LIN {X 0,Y 474.559,Z 355.992,A -85,B 0,C 180,E1 -7422.941,E2 -7422.941} C_VEL
LIN {X 0,Y 474.594,Z 355.995,A -85,B 0,C 180,E1 -7425.896,E2 -7425.896} C_VEL
LIN {X 0,Y 474.593,Z 355.988,A -85,B 0,C 180,E1 -7429.046,E2 -7429.046} C_VEL
LIN {X 0,Y 474.585,Z 355.996,A -85,B 0,C 180,E1 -7431.708,E2 -7431.708} C_VEL
LIN {X 0,Y 474.612,Z 355.985,A -85,B 0,C 180,E1 -7434.727,E2 -7434.727} C_VEL
LIN {X 0,Y 474.63,Z 355.992,A -85,B 0,C 180,E1 -7437.789,E2 -7437.789} C_VEL
LIN {X 0,Y 474.593,Z 355.988,A -85,B 0,C 180,E1 -7440.892,E2 -7440.892} C_VEL
LIN {X 0,Y 474.579,Z 355.996,A -85,B 0,C 180,E1 -7443.625,E2 -7443.625} C_VEL
LIN {X 0,Y 474.632,Z 355.983,A -85,B 0,C 180,E1 -7446.644,E2 -7446.644} C_VEL
LIN {X 0,Y 474.65,Z 355.984,A -85,B 0,C 180,E1 -7450.091,E2 -7450.091} C_VEL
LIN {X 0,Y 474.642,Z 355.986,A -85,B 0,C 180,E1 -7451.641,E2 -7451.641} C_VEL
LIN {X 0,Y 473.97,Z 356.072,A -85,B 0,C 180,E1 -7452.35,E2 -7452.35} C_VEL
LIN {X 0,Y 471.124,Z 356.427,A -85,B 0,C 180,E1 -7453.501,E2 -7453.501} C_VEL
LIN {X 0,Y 468.718,Z 356.724,A -85,B 0,C 180,E1 -7454.429,E2 -7454.429} C_VEL
LIN {X 0,Y 467.679,Z 356.851,A -85,B 0,C 180,E1 -7455.147,E2 -7455.147} C_VEL
LIN {X 0,Y 467.592,Z 356.861,A -85,B 0,C 180,E1 -7455.389,E2 -7455.389} C_VEL
LIN {X 0,Y 467.65,Z 356.853,A -85,B 0,C 180,E1 -7458.735,E2 -7458.735} C_VEL
LIN {X 0,Y 467.658,Z 356.855,A -85,B 0,C 180,E1 -7461.358,E2 -7461.358} C_VEL
LIN {X 0,Y 467.705,Z 356.85,A -85,B 0,C 180,E1 -7463.963,E2 -7463.963} C_VEL
LIN {X 0,Y 467.816,Z 356.837,A -85,B 0,C 180,E1 -7467.418,E2 -7467.418} C_VEL
LIN {X 0,Y 467.853,Z 356.831,A -85,B 0,C 180,E1 -7470.001,E2 -7470.001} C_VEL
LIN {X 0,Y 467.818,Z 356.832,A -85,B 0,C 180,E1 -7472.584,E2 -7472.584} C_VEL
LIN {X 0,Y 467.708,Z 356.848,A -85,B 0,C 180,E1 -7476.039,E2 -7476.039} C_VEL
LIN {X 0,Y 467.671,Z 356.85,A -85,B 0,C 180,E1 -7478.644,E2 -7478.644} C_VEL
LIN {X 0,Y 467.662,Z 356.853,A -85,B 0,C 180,E1 -7482.146,E2 -7482.146} C_VEL
LIN {X 0,Y 467.618,Z 356.864,A -85,B 0,C 180,E1 -7485.697,E2 -7485.697} C_VEL
LIN {X 0,Y 467.626,Z 356.86,A -85,B 0,C 180,E1 -7489.309,E2 -7489.309} C_VEL
LIN {X 0,Y 467.54,Z 356.868,A -85,B 0,C 180,E1 -7492.075,E2 -7492.075} C_VEL
LIN {X 0,Y 467.565,Z 356.864,A -85,B 0,C 180,E1 -7494.891,E2 -7494.891} C_VEL
LIN {X 0,Y 467.552,Z 356.87,A -85,B 0,C 180,E1 -7497.774,E2 -7497.774} C_VEL
LIN {X 0,Y 467.572,Z 356.865,A -85,B 0,C 180,E1 -7501.045,E2 -7501.045} C_VEL
LIN {X 0,Y 467.593,Z 356.86,A -85,B 0,C 180,E1 -7504.242,E2 -7504.242} C_VEL
LIN {X 0,Y 467.549,Z 356.873,A -85,B 0,C 180,E1 -7507.186,E2 -7507.186} C_VEL
LIN {X 0,Y 467.576,Z 356.867,A -85,B 0,C 180,E1 -7510.266,E2 -7510.266} C_VEL
LIN {X 0,Y 467.567,Z 356.868,A -85,B 0,C 180,E1 -7512.564,E2 -7512.564} C_VEL
LIN {X 0,Y 467.561,Z 356.872,A -85,B 0,C 180,E1 -7514.121,E2 -7514.121} C_VEL
LIN {X 0,Y 470.952,Z 371.96,A -85,B 0,C 180,E1 -7516.951,E2 -7516.951} C_VEL
LIN {X 0,Y 474.676,Z 387.334,A -85,B 0,C 180,E1 -7517.428,E2 -7517.428} C_VEL
LIN {X 0,Y 475.85,Z 392.656,A -85,B 0,C 180,E1 -7517.582,E2 -7517.582} C_VEL
LIN {X 0,Y 473.727,Z 537.942,A -85,B 0,C 180,E1 -7519.999,E2 -7519.999} C_VEL
LIN {X 0,Y 473.257,Z 553.297,A -85,B 0,C 180,E1 -7520.424,E2 -7520.424} C_VEL
LIN {X 0,Y 472.684,Z 567.565,A -85,B 0,C 180,E1 -7520.982,E2 -7520.982} C_VEL
LIN {X 0,Y 471.947,Z 582.804,A -85,B 0,C 180,E1 -7521.773,E2 -7521.773} C_VEL
LIN {X 0,Y 471.223,Z 596.937,A -85,B 0,C 180,E1 -7522.706,E2 -7522.706} C_VEL
LIN {X 0,Y 470.38,Z 610.271,A -85,B 0,C 180,E1 -7523.788,E2 -7523.788} C_VEL
LIN {X 0,Y 469.675,Z 622.164,A -85,B 0,C 180,E1 -7524.954,E2 -7524.954} C_VEL
LIN {X 0,Y 468.906,Z 633.77,A -85,B 0,C 180,E1 -7526.319,E2 -7526.319} C_VEL
LIN {X 0,Y 468.273,Z 644.266,A -85,B 0,C 180,E1 -7527.805,E2 -7527.805} C_VEL
LIN {X 0,Y 467.78,Z 652.986,A -85,B 0,C 180,E1 -7529.281,E2 -7529.281} C_VEL
LIN {X 0,Y 467.331,Z 661.21,A -85,B 0,C 180,E1 -7530.971,E2 -7530.971} C_VEL
LIN {X 0,Y 467.022,Z 667.684,A -85,B 0,C 180,E1 -7532.607,E2 -7532.607} C_VEL
LIN {X 0,Y 466.836,Z 672.428,A -85,B 0,C 180,E1 -7534.114,E2 -7534.114} C_VEL
LIN {X 0,Y 466.715,Z 676.016,A -85,B 0,C 180,E1 -7535.537,E2 -7535.537} C_VEL
LIN {X 0,Y 466.612,Z 678.697,A -85,B 0,C 180,E1 -7536.945,E2 -7536.945} C_VEL
LIN {X 0,Y 466.538,Z 681.023,A -85,B 0,C 180,E1 -7538.805,E2 -7538.805} C_VEL
LIN {X 0,Y 466.523,Z 681.987,A -85,B 0,C 180,E1 -7540.645,E2 -7540.645} C_VEL
LIN {X 0,Y 466.534,Z 681.648,A -85,B 0,C 180,E1 -7542.465,E2 -7542.465} C_VEL
LIN {X 0,Y 466.539,Z 680.045,A -85,B 0,C 180,E1 -7544.267,E2 -7544.267} C_VEL
LIN {X 0,Y 466.613,Z 677.173,A -85,B 0,C 180,E1 -7546.055,E2 -7546.055} C_VEL
LIN {X 0,Y 466.856,Z 672.982,A -85,B 0,C 180,E1 -7547.833,E2 -7547.833} C_VEL
LIN {X 0,Y 467.035,Z 667.435,A -85,B 0,C 180,E1 -7549.596,E2 -7549.596} C_VEL
LIN {X 0,Y 467.402,Z 660.369,A -85,B 0,C 180,E1 -7551.352,E2 -7551.352} C_VEL
LIN {X 0,Y 467.801,Z 653.127,A -85,B 0,C 180,E1 -7552.824,E2 -7552.824} C_VEL
LIN {X 0,Y 468.295,Z 643.765,A -85,B 0,C 180,E1 -7554.402,E2 -7554.402} C_VEL
LIN {X 0,Y 468.97,Z 632.863,A -85,B 0,C 180,E1 -7555.918,E2 -7555.918} C_VEL
LIN {X 0,Y 469.723,Z 621.677,A -85,B 0,C 180,E1 -7557.213,E2 -7557.213} C_VEL
LIN {X 0,Y 470.482,Z 609.45,A -85,B 0,C 180,E1 -7558.395,E2 -7558.395} C_VEL
LIN {X 0,Y 471.319,Z 596.43,A -85,B 0,C 180,E1 -7559.435,E2 -7559.435} C_VEL
LIN {X 0,Y 472.012,Z 582.911,A -85,B 0,C 180,E1 -7560.32,E2 -7560.32} C_VEL
LIN {X 0,Y 472.671,Z 568.576,A -85,B 0,C 180,E1 -7561.065,E2 -7561.065} C_VEL
LIN {X 0,Y 473.286,Z 552.999,A -85,B 0,C 180,E1 -7561.675,E2 -7561.675} C_VEL
LIN {X 0,Y 473.757,Z 537.298,A -85,B 0,C 180,E1 -7562.099,E2 -7562.099} C_VEL
LIN {X 0,Y 476.168,Z 392.734,A -85,B 0,C 180,E1 -7564.596,E2 -7564.596} C_VEL
LIN {X 0,Y 472.006,Z 375.11,A -85,B 0,C 180,E1 -7565.179,E2 -7565.179} C_VEL
LIN {X 0,Y 471.448,Z 373.4,A -85,B 0,C 180,E1 -7565.265,E2 -7565.265} C_VEL
LIN {X 0,Y 469.366,Z 363.6,A -85,B 0,C 180,E1 -7567.194,E2 -7567.194} C_VEL
LIN {X 0,Y 467.682,Z 356.858,A -85,B 0,C 180,E1 -7568.613,E2 -7568.613} C_VEL
LIN {X 0,Y 467.661,Z 356.858,A -85,B 0,C 180,E1 -7572.145,E2 -7572.145} C_VEL
LIN {X 0,Y 467.643,Z 356.859,A -85,B 0,C 180,E1 -7575.695,E2 -7575.695} C_VEL
LIN {X 0,Y 467.626,Z 356.86,A -85,B 0,C 180,E1 -7579.307,E2 -7579.307} C_VEL
LIN {X 0,Y 467.539,Z 356.873,A -85,B 0,C 180,E1 -7582.073,E2 -7582.073} C_VEL
LIN {X 0,Y 467.559,Z 356.867,A -85,B 0,C 180,E1 -7584.89,E2 -7584.89} C_VEL
LIN {X 0,Y 467.548,Z 356.871,A -85,B 0,C 180,E1 -7587.773,E2 -7587.773} C_VEL
LIN {X 0,Y 467.55,Z 356.867,A -85,B 0,C 180,E1 -7591.04,E2 -7591.04} C_VEL
LIN {X 0,Y 467.578,Z 356.868,A -85,B 0,C 180,E1 -7594.239,E2 -7594.239} C_VEL
LIN {X 0,Y 467.517,Z 356.872,A -85,B 0,C 180,E1 -7597.18,E2 -7597.18} C_VEL
LIN {X 0,Y 467.541,Z 356.872,A -85,B 0,C 180,E1 -7600.268,E2 -7600.268} C_VEL
LIN {X 0,Y 467.519,Z 356.873,A -85,B 0,C 180,E1 -7602.568,E2 -7602.568} C_VEL
LIN {X 0,Y 467.564,Z 356.864,A -85,B 0,C 180,E1 -7605.051,E2 -7605.051} C_VEL
LIN {X 0,Y 467.552,Z 356.867,A -85,B 0,C 180,E1 -7608.727,E2 -7608.727} C_VEL
LIN {X 0,Y 467.539,Z 356.875,A -85,B 0,C 180,E1 -7611.952,E2 -7611.952} C_VEL
LIN {X 0,Y 467.541,Z 356.873,A -85,B 0,C 180,E1 -7615.164,E2 -7615.164} C_VEL
LIN {X 0,Y 467.551,Z 356.877,A -85,B 0,C 180,E1 -7618.256,E2 -7618.256} C_VEL
LIN {X 0,Y 467.609,Z 356.988,A -85,B 0,C 180,E1 -7619.362,E2 -7619.362} C_VEL
LIN {X 0,Y 470.846,Z 369.937,A -85,B 0,C 180,E1 -7621.721,E2 -7621.721} C_VEL
LIN {X 0,Y 472.31,Z 377.176,A -85,B 0,C 180,E1 -7622.965,E2 -7622.965} C_VEL
LIN {X 0,Y 471.285,Z 396.039,A -85,B 0,C 180,E1 -7625.777,E2 -7625.777} C_VEL
LIN {X 0,Y 475.861,Z 420.157,A -85,B 0,C 180,E1 -7626.498,E2 -7626.498} C_VEL
LIN {X 0,Y 474.004,Z 533.469,A -85,B 0,C 180,E1 -7628.442,E2 -7628.442} C_VEL
LIN {X 0,Y 473.478,Z 564.563,A -85,B 0,C 180,E1 -7628.987,E2 -7628.987} C_VEL
LIN {X 0,Y 472.916,Z 580.082,A -85,B 0,C 180,E1 -7629.429,E2 -7629.429} C_VEL
LIN {X 0,Y 472.302,Z 595.204,A -85,B 0,C 180,E1 -7630.042,E2 -7630.042} C_VEL
LIN {X 0,Y 471.659,Z 608.713,A -85,B 0,C 180,E1 -7630.75,E2 -7630.75} C_VEL
LIN {X 0,Y 470.924,Z 622.125,A -85,B 0,C 180,E1 -7631.622,E2 -7631.622} C_VEL
LIN {X 0,Y 470.114,Z 634.534,A -85,B 0,C 180,E1 -7632.602,E2 -7632.602} C_VEL
LIN {X 0,Y 469.374,Z 647.182,A -85,B 0,C 180,E1 -7633.806,E2 -7633.806} C_VEL
LIN {X 0,Y 468.596,Z 659.56,A -85,B 0,C 180,E1 -7635.227,E2 -7635.227} C_VEL
LIN {X 0,Y 468.049,Z 669.126,A -85,B 0,C 180,E1 -7636.54,E2 -7636.54} C_VEL
LIN {X 0,Y 467.526,Z 678.506,A -85,B 0,C 180,E1 -7638.07,E2 -7638.07} C_VEL
LIN {X 0,Y 467.224,Z 686.288,A -85,B 0,C 180,E1 -7639.6,E2 -7639.6} C_VEL
LIN {X 0,Y 466.907,Z 693.544,A -85,B 0,C 180,E1 -7641.342,E2 -7641.342} C_VEL
LIN {X 0,Y 466.745,Z 699.247,A -85,B 0,C 180,E1 -7643.08,E2 -7643.08} C_VEL
LIN {X 0,Y 466.686,Z 703.56,A -85,B 0,C 180,E1 -7644.815,E2 -7644.815} C_VEL
LIN {X 0,Y 466.639,Z 706.587,A -85,B 0,C 180,E1 -7646.545,E2 -7646.545} C_VEL
LIN {X 0,Y 466.628,Z 708.398,A -85,B 0,C 180,E1 -7648.273,E2 -7648.273} C_VEL
LIN {X 0,Y 466.595,Z 709.029,A -85,B 0,C 180,E1 -7649.999,E2 -7649.999} C_VEL
LIN {X 0,Y 466.628,Z 708.435,A -85,B 0,C 180,E1 -7651.725,E2 -7651.725} C_VEL
LIN {X 0,Y 466.67,Z 706.662,A -85,B 0,C 180,E1 -7653.452,E2 -7653.452} C_VEL
LIN {X 0,Y 466.69,Z 703.683,A -85,B 0,C 180,E1 -7655.183,E2 -7655.183} C_VEL
LIN {X 0,Y 466.82,Z 699.43,A -85,B 0,C 180,E1 -7656.916,E2 -7656.916} C_VEL
LIN {X 0,Y 466.933,Z 693.785,A -85,B 0,C 180,E1 -7658.655,E2 -7658.655} C_VEL
LIN {X 0,Y 467.222,Z 686.598,A -85,B 0,C 180,E1 -7660.398,E2 -7660.398} C_VEL
LIN {X 0,Y 467.601,Z 678.901,A -85,B 0,C 180,E1 -7661.925,E2 -7661.925} C_VEL
LIN {X 0,Y 468.081,Z 669.621,A -85,B 0,C 180,E1 -7663.456,E2 -7663.456} C_VEL
LIN {X 0,Y 468.648,Z 660.149,A -85,B 0,C 180,E1 -7664.768,E2 -7664.768} C_VEL
LIN {X 0,Y 469.455,Z 647.921,A -85,B 0,C 180,E1 -7666.189,E2 -7666.189} C_VEL
LIN {X 0,Y 470.178,Z 635.42,A -85,B 0,C 180,E1 -7667.393,E2 -7667.393} C_VEL
LIN {X 0,Y 470.931,Z 623.112,A -85,B 0,C 180,E1 -7668.375,E2 -7668.375} C_VEL
LIN {X 0,Y 471.738,Z 609.861,A -85,B 0,C 180,E1 -7669.244,E2 -7669.244} C_VEL
LIN {X 0,Y 472.39,Z 596.536,A -85,B 0,C 180,E1 -7669.952,E2 -7669.952} C_VEL
LIN {X 0,Y 473.025,Z 581.741,A -85,B 0,C 180,E1 -7670.56,E2 -7670.56} C_VEL
LIN {X 0,Y 473.553,Z 566.453,A -85,B 0,C 180,E1 -7671.007,E2 -7671.007} C_VEL
LIN {X 0,Y 473.94,Z 543.805,A -85,B 0,C 180,E1 -7671.416,E2 -7671.416} C_VEL
LIN {X 0,Y 475.645,Z 419.81,A -85,B 0,C 180,E1 -7673.463,E2 -7673.463} C_VEL
LIN {X 0,Y 471.258,Z 396.949,A -85,B 0,C 180,E1 -7674.105,E2 -7674.105} C_VEL
LIN {X 0,Y 472.297,Z 378.855,A -85,B 0,C 180,E1 -7676.77,E2 -7676.77} C_VEL
LIN {X 0,Y 472.051,Z 375.647,A -85,B 0,C 180,E1 -7677.27,E2 -7677.27} C_VEL
LIN {X 0,Y 468.726,Z 361.5,A -85,B 0,C 180,E1 -7679.654,E2 -7679.654} C_VEL
LIN {X 0,Y 467.582,Z 356.868,A -85,B 0,C 180,E1 -7680.481,E2 -7680.481} C_VEL
LIN {X 0,Y 467.561,Z 356.869,A -85,B 0,C 180,E1 -7683.788,E2 -7683.788} C_VEL
LIN {X 0,Y 467.503,Z 356.874,A -85,B 0,C 180,E1 -7686.963,E2 -7686.963} C_VEL
LIN {X 0,Y 467.551,Z 356.871,A -85,B 0,C 180,E1 -7689.95,E2 -7689.95} C_VEL
LIN {X 0,Y 467.532,Z 356.871,A -85,B 0,C 180,E1 -7692.564,E2 -7692.564} C_VEL
LIN {X 0,Y 467.553,Z 356.865,A -85,B 0,C 180,E1 -7695.051,E2 -7695.051} C_VEL
LIN {X 0,Y 467.548,Z 356.867,A -85,B 0,C 180,E1 -7698.725,E2 -7698.725} C_VEL
LIN {X 0,Y 467.528,Z 356.873,A -85,B 0,C 180,E1 -7701.952,E2 -7701.952} C_VEL
LIN {X 0,Y 467.544,Z 356.866,A -85,B 0,C 180,E1 -7705.166,E2 -7705.166} C_VEL
LIN {X 0,Y 467.568,Z 356.87,A -85,B 0,C 180,E1 -7708.259,E2 -7708.259} C_VEL
LIN {X 0,Y 467.529,Z 356.868,A -85,B 0,C 180,E1 -7711.247,E2 -7711.247} C_VEL
LIN {X 0,Y 467.563,Z 356.868,A -85,B 0,C 180,E1 -7714.4,E2 -7714.4} C_VEL
LIN {X 0,Y 467.556,Z 356.864,A -85,B 0,C 180,E1 -7716.995,E2 -7716.995} C_VEL
LIN {X 0,Y 467.604,Z 356.863,A -85,B 0,C 180,E1 -7719.777,E2 -7719.777} C_VEL
LIN {X 0,Y 467.55,Z 356.868,A -85,B 0,C 180,E1 -7722.505,E2 -7722.505} C_VEL
LIN {X 0,Y 467.577,Z 356.862,A -85,B 0,C 180,E1 -7725.196,E2 -7725.196} C_VEL
LIN {X 0,Y 467.64,Z 356.859,A -85,B 0,C 180,E1 -7727.854,E2 -7727.854} C_VEL
LIN {X 0,Y 467.641,Z 356.855,A -85,B 0,C 180,E1 -7731.357,E2 -7731.357} C_VEL
LIN {X 0,Y 467.69,Z 356.855,A -85,B 0,C 180,E1 -7733.962,E2 -7733.962} C_VEL
LIN {X 0,Y 467.796,Z 356.836,A -85,B 0,C 180,E1 -7737.417,E2 -7737.417} C_VEL
LIN {X 0,Y 467.833,Z 356.838,A -85,B 0,C 180,E1 -7740,E2 -7740} C_VEL
LIN {X 0,Y 467.796,Z 356.836,A -85,B 0,C 180,E1 -7742.583,E2 -7742.583} C_VEL
LIN {X 0,Y 467.686,Z 356.856,A -85,B 0,C 180,E1 -7746.038,E2 -7746.038} C_VEL
LIN {X 0,Y 467.639,Z 356.855,A -85,B 0,C 180,E1 -7748.644,E2 -7748.644} C_VEL
LIN {X 0,Y 467.633,Z 356.858,A -85,B 0,C 180,E1 -7752.354,E2 -7752.354} C_VEL
LIN {X 0,Y 467.585,Z 356.868,A -85,B 0,C 180,E1 -7755.864,E2 -7755.864} C_VEL
LIN {X 0,Y 467.604,Z 356.86,A -85,B 0,C 180,E1 -7759.309,E2 -7759.309} C_VEL
LIN {X 0,Y 467.516,Z 356.876,A -85,B 0,C 180,E1 -7762.075,E2 -7762.075} C_VEL
LIN {X 0,Y 467.545,Z 356.866,A -85,B 0,C 180,E1 -7764.891,E2 -7764.891} C_VEL
LIN {X 0,Y 467.531,Z 356.874,A -85,B 0,C 180,E1 -7767.775,E2 -7767.775} C_VEL
LIN {X 0,Y 467.553,Z 356.865,A -85,B 0,C 180,E1 -7771.045,E2 -7771.045} C_VEL
LIN {X 0,Y 467.565,Z 356.867,A -85,B 0,C 180,E1 -7774.241,E2 -7774.241} C_VEL
LIN {X 0,Y 467.506,Z 356.871,A -85,B 0,C 180,E1 -7777.183,E2 -7777.183} C_VEL
LIN {X 0,Y 467.546,Z 356.868,A -85,B 0,C 180,E1 -7780.268,E2 -7780.268} C_VEL
LIN {X 0,Y 467.535,Z 356.874,A -85,B 0,C 180,E1 -7783.747,E2 -7783.747} C_VEL
LIN {X 0,Y 467.538,Z 356.869,A -85,B 0,C 180,E1 -7786.256,E2 -7786.256} C_VEL
LIN {X 0,Y 467.549,Z 356.873,A -85,B 0,C 180,E1 -7789.735,E2 -7789.735} C_VEL
LIN {X 0,Y 467.516,Z 356.869,A -85,B 0,C 180,E1 -7792.82,E2 -7792.82} C_VEL
LIN {X 0,Y 467.571,Z 356.871,A -85,B 0,C 180,E1 -7795.762,E2 -7795.762} C_VEL
LIN {X 0,Y 467.561,Z 356.864,A -85,B 0,C 180,E1 -7798.957,E2 -7798.957} C_VEL
LIN {X 0,Y 467.54,Z 356.869,A -85,B 0,C 180,E1 -7802.228,E2 -7802.228} C_VEL
LIN {X 0,Y 467.553,Z 356.866,A -85,B 0,C 180,E1 -7805.112,E2 -7805.112} C_VEL
LIN {X 0,Y 467.533,Z 356.873,A -85,B 0,C 180,E1 -7807.928,E2 -7807.928} C_VEL
LIN {X 0,Y 467.619,Z 356.856,A -85,B 0,C 180,E1 -7810.694,E2 -7810.694} C_VEL
LIN {X 0,Y 467.638,Z 356.856,A -85,B 0,C 180,E1 -7814.306,E2 -7814.306} C_VEL
LIN {X 0,Y 467.592,Z 356.861,A -85,B 0,C 180,E1 -7815.389,E2 -7815.389} C_VEL
LIN {X 0,Y 466.92,Z 356.947,A -85,B 0,C 180,E1 -7816.109,E2 -7816.109} C_VEL
LIN {X 0,Y 464.081,Z 357.3,A -85,B 0,C 180,E1 -7817.277,E2 -7817.277} C_VEL
LIN {X 0,Y 461.684,Z 357.598,A -85,B 0,C 180,E1 -7818.22,E2 -7818.22} C_VEL
LIN {X 0,Y 460.656,Z 357.725,A -85,B 0,C 180,E1 -7818.947,E2 -7818.947} C_VEL
LIN {X 0,Y 460.572,Z 357.736,A -85,B 0,C 180,E1 -7819.194,E2 -7819.194} C_VEL
LIN {X 0,Y 460.665,Z 357.723,A -85,B 0,C 180,E1 -7822.595,E2 -7822.595} C_VEL
LIN {X 0,Y 460.677,Z 357.721,A -85,B 0,C 180,E1 -7824.749,E2 -7824.749} C_VEL
LIN {X 0,Y 460.76,Z 357.715,A -85,B 0,C 180,E1 -7827.379,E2 -7827.379} C_VEL
LIN {X 0,Y 460.822,Z 357.707,A -85,B 0,C 180,E1 -7830.001,E2 -7830.001} C_VEL
LIN {X 0,Y 460.762,Z 357.711,A -85,B 0,C 180,E1 -7832.624,E2 -7832.624} C_VEL
LIN {X 0,Y 460.674,Z 357.724,A -85,B 0,C 180,E1 -7836.132,E2 -7836.132} C_VEL
LIN {X 0,Y 460.622,Z 357.728,A -85,B 0,C 180,E1 -7838.777,E2 -7838.777} C_VEL
LIN {X 0,Y 460.602,Z 357.731,A -85,B 0,C 180,E1 -7842.436,E2 -7842.436} C_VEL
LIN {X 0,Y 460.562,Z 357.739,A -85,B 0,C 180,E1 -7845.979,E2 -7845.979} C_VEL
LIN {X 0,Y 460.572,Z 357.742,A -85,B 0,C 180,E1 -7849.616,E2 -7849.616} C_VEL
LIN {X 0,Y 460.516,Z 357.741,A -85,B 0,C 180,E1 -7852.43,E2 -7852.43} C_VEL
LIN {X 0,Y 460.541,Z 357.743,A -85,B 0,C 180,E1 -7855.794,E2 -7855.794} C_VEL
LIN {X 0,Y 460.526,Z 357.744,A -85,B 0,C 180,E1 -7859.233,E2 -7859.233} C_VEL
LIN {X 0,Y 460.537,Z 357.739,A -85,B 0,C 180,E1 -7862.285,E2 -7862.285} C_VEL
LIN {X 0,Y 460.514,Z 357.749,A -85,B 0,C 180,E1 -7865.446,E2 -7865.446} C_VEL
LIN {X 0,Y 460.511,Z 357.747,A -85,B 0,C 180,E1 -7868.892,E2 -7868.892} C_VEL
LIN {X 0,Y 460.524,Z 357.748,A -85,B 0,C 180,E1 -7871.601,E2 -7871.601} C_VEL
LIN {X 0,Y 460.523,Z 357.748,A -85,B 0,C 180,E1 -7873.827,E2 -7873.827} C_VEL
LIN {X 0,Y 463.793,Z 372.282,A -85,B 0,C 180,E1 -7876.587,E2 -7876.587} C_VEL
LIN {X 0,Y 465.856,Z 378.515,A -85,B 0,C 180,E1 -7876.813,E2 -7876.813} C_VEL
LIN {X 0,Y 469.226,Z 393.41,A -85,B 0,C 180,E1 -7877.256,E2 -7877.256} C_VEL
LIN {X 0,Y 467.185,Z 529.999,A -85,B 0,C 180,E1 -7879.553,E2 -7879.553} C_VEL
LIN {X 0,Y 466.793,Z 546.261,A -85,B 0,C 180,E1 -7879.92,E2 -7879.92} C_VEL
LIN {X 0,Y 466.209,Z 561.626,A -85,B 0,C 180,E1 -7880.448,E2 -7880.448} C_VEL
LIN {X 0,Y 465.578,Z 576.36,A -85,B 0,C 180,E1 -7881.141,E2 -7881.141} C_VEL
LIN {X 0,Y 464.891,Z 589.468,A -85,B 0,C 180,E1 -7881.921,E2 -7881.921} C_VEL
LIN {X 0,Y 463.999,Z 603.248,A -85,B 0,C 180,E1 -7882.933,E2 -7882.933} C_VEL
LIN {X 0,Y 463.243,Z 615.11,A -85,B 0,C 180,E1 -7883.992,E2 -7883.992} C_VEL
LIN {X 0,Y 462.492,Z 625.965,A -85,B 0,C 180,E1 -7885.144,E2 -7885.144} C_VEL
LIN {X 0,Y 461.744,Z 636.861,A -85,B 0,C 180,E1 -7886.513,E2 -7886.513} C_VEL
LIN {X 0,Y 461.153,Z 646.802,A -85,B 0,C 180,E1 -7888.008,E2 -7888.008} C_VEL
LIN {X 0,Y 460.63,Z 655.174,A -85,B 0,C 180,E1 -7889.515,E2 -7889.515} C_VEL
LIN {X 0,Y 460.228,Z 663.103,A -85,B 0,C 180,E1 -7891.247,E2 -7891.247} C_VEL
LIN {X 0,Y 459.941,Z 668.61,A -85,B 0,C 180,E1 -7892.715,E2 -7892.715} C_VEL
LIN {X 0,Y 459.74,Z 673.716,A -85,B 0,C 180,E1 -7894.414,E2 -7894.414} C_VEL
LIN {X 0,Y 459.625,Z 676.526,A -85,B 0,C 180,E1 -7895.616,E2 -7895.616} C_VEL
LIN {X 0,Y 459.453,Z 679.82,A -85,B 0,C 180,E1 -7897.517,E2 -7897.517} C_VEL
LIN {X 0,Y 459.448,Z 681.698,A -85,B 0,C 180,E1 -7899.401,E2 -7899.401} C_VEL
LIN {X 0,Y 459.444,Z 682.236,A -85,B 0,C 180,E1 -7901.262,E2 -7901.262} C_VEL
LIN {X 0,Y 459.428,Z 681.484,A -85,B 0,C 180,E1 -7903.103,E2 -7903.103} C_VEL
LIN {X 0,Y 459.505,Z 679.461,A -85,B 0,C 180,E1 -7904.929,E2 -7904.929} C_VEL
LIN {X 0,Y 459.624,Z 676.139,A -85,B 0,C 180,E1 -7906.74,E2 -7906.74} C_VEL
LIN {X 0,Y 459.823,Z 671.486,A -85,B 0,C 180,E1 -7908.539,E2 -7908.539} C_VEL
LIN {X 0,Y 460.074,Z 665.437,A -85,B 0,C 180,E1 -7910.326,E2 -7910.326} C_VEL
LIN {X 0,Y 460.531,Z 657.824,A -85,B 0,C 180,E1 -7912.105,E2 -7912.105} C_VEL
LIN {X 0,Y 461.003,Z 649.687,A -85,B 0,C 180,E1 -7913.654,E2 -7913.654} C_VEL
LIN {X 0,Y 461.624,Z 639.949,A -85,B 0,C 180,E1 -7915.196,E2 -7915.196} C_VEL
LIN {X 0,Y 462.315,Z 630.001,A -85,B 0,C 180,E1 -7916.514,E2 -7916.514} C_VEL
LIN {X 0,Y 463.062,Z 618.257,A -85,B 0,C 180,E1 -7917.825,E2 -7917.825} C_VEL
LIN {X 0,Y 463.929,Z 605.963,A -85,B 0,C 180,E1 -7918.964,E2 -7918.964} C_VEL
LIN {X 0,Y 464.735,Z 592.437,A -85,B 0,C 180,E1 -7920,E2 -7920} C_VEL
LIN {X 0,Y 465.533,Z 578.411,A -85,B 0,C 180,E1 -7920.865,E2 -7920.865} C_VEL
LIN {X 0,Y 466.188,Z 563.974,A -85,B 0,C 180,E1 -7921.566,E2 -7921.566} C_VEL
LIN {X 0,Y 466.749,Z 549.143,A -85,B 0,C 180,E1 -7922.103,E2 -7922.103} C_VEL
LIN {X 0,Y 467.168,Z 533.927,A -85,B 0,C 180,E1 -7922.479,E2 -7922.479} C_VEL
LIN {X 0,Y 469.596,Z 402.99,A -85,B 0,C 180,E1 -7924.781,E2 -7924.781} C_VEL
LIN {X 0,Y 469.695,Z 393.427,A -85,B 0,C 180,E1 -7924.963,E2 -7924.963} C_VEL
LIN {X 0,Y 465.864,Z 377.43,A -85,B 0,C 180,E1 -7925.518,E2 -7925.518} C_VEL
LIN {X 0,Y 464.428,Z 373.801,A -85,B 0,C 180,E1 -7925.684,E2 -7925.684} C_VEL
LIN {X 0,Y 462.015,Z 363.103,A -85,B 0,C 180,E1 -7927.869,E2 -7927.869} C_VEL
LIN {X 0,Y 460.636,Z 357.734,A -85,B 0,C 180,E1 -7929.052,E2 -7929.052} C_VEL
LIN {X 0,Y 460.602,Z 357.737,A -85,B 0,C 180,E1 -7932.435,E2 -7932.435} C_VEL
LIN {X 0,Y 460.606,Z 357.738,A -85,B 0,C 180,E1 -7935.997,E2 -7935.997} C_VEL
LIN {X 0,Y 460.572,Z 357.739,A -85,B 0,C 180,E1 -7939.615,E2 -7939.615} C_VEL
LIN {X 0,Y 460.515,Z 357.749,A -85,B 0,C 180,E1 -7942.428,E2 -7942.428} C_VEL
LIN {X 0,Y 460.536,Z 357.743,A -85,B 0,C 180,E1 -7945.792,E2 -7945.792} C_VEL
LIN {X 0,Y 460.522,Z 357.744,A -85,B 0,C 180,E1 -7949.232,E2 -7949.232} C_VEL
LIN {X 0,Y 460.521,Z 357.748,A -85,B 0,C 180,E1 -7952.285,E2 -7952.285} C_VEL
LIN {X 0,Y 460.502,Z 357.747,A -85,B 0,C 180,E1 -7955.446,E2 -7955.446} C_VEL
LIN {X 0,Y 460.486,Z 357.747,A -85,B 0,C 180,E1 -7958.887,E2 -7958.887} C_VEL
LIN {X 0,Y 460.497,Z 357.748,A -85,B 0,C 180,E1 -7961.596,E2 -7961.596} C_VEL
LIN {X 0,Y 460.508,Z 357.744,A -85,B 0,C 180,E1 -7964.589,E2 -7964.589} C_VEL
LIN {X 0,Y 460.473,Z 357.752,A -85,B 0,C 180,E1 -7967.812,E2 -7967.812} C_VEL
LIN {X 0,Y 460.477,Z 357.752,A -85,B 0,C 180,E1 -7970.131,E2 -7970.131} C_VEL
LIN {X 0,Y 460.458,Z 357.756,A -85,B 0,C 180,E1 -7973.468,E2 -7973.468} C_VEL
LIN {X 0,Y 460.503,Z 357.753,A -85,B 0,C 180,E1 -7976.672,E2 -7976.672} C_VEL
LIN {X 0,Y 460.519,Z 357.849,A -85,B 0,C 180,E1 -7978.934,E2 -7978.934} C_VEL
LIN {X 0,Y 463.633,Z 369.945,A -85,B 0,C 180,E1 -7981.216,E2 -7981.216} C_VEL
LIN {X 0,Y 465.571,Z 379.235,A -85,B 0,C 180,E1 -7982.853,E2 -7982.853} C_VEL
LIN {X 0,Y 464.544,Z 395.515,A -85,B 0,C 180,E1 -7985.349,E2 -7985.349} C_VEL
LIN {X 0,Y 469.424,Z 421.293,A -85,B 0,C 180,E1 -7986.156,E2 -7986.156} C_VEL
LIN {X 0,Y 467.381,Z 534.879,A -85,B 0,C 180,E1 -7988.15,E2 -7988.15} C_VEL
LIN {X 0,Y 466.861,Z 564.068,A -85,B 0,C 180,E1 -7988.675,E2 -7988.675} C_VEL
LIN {X 0,Y 466.286,Z 579.38,A -85,B 0,C 180,E1 -7989.115,E2 -7989.115} C_VEL
LIN {X 0,Y 465.594,Z 594.743,A -85,B 0,C 180,E1 -7989.742,E2 -7989.742} C_VEL
LIN {X 0,Y 464.896,Z 608.292,A -85,B 0,C 180,E1 -7990.458,E2 -7990.458} C_VEL
LIN {X 0,Y 464.115,Z 621.72,A -85,B 0,C 180,E1 -7991.343,E2 -7991.343} C_VEL
LIN {X 0,Y 463.177,Z 635.394,A -85,B 0,C 180,E1 -7992.447,E2 -7992.447} C_VEL
LIN {X 0,Y 462.399,Z 647.848,A -85,B 0,C 180,E1 -7993.668,E2 -7993.668} C_VEL
LIN {X 0,Y 461.619,Z 659.226,A -85,B 0,C 180,E1 -7994.999,E2 -7994.999} C_VEL
LIN {X 0,Y 461.061,Z 668.805,A -85,B 0,C 180,E1 -7996.332,E2 -7996.332} C_VEL
LIN {X 0,Y 460.504,Z 678.203,A -85,B 0,C 180,E1 -7997.885,E2 -7997.885} C_VEL
LIN {X 0,Y 460.202,Z 686.012,A -85,B 0,C 180,E1 -7999.439,E2 -7999.439} C_VEL
LIN {X 0,Y 459.851,Z 693.286,A -85,B 0,C 180,E1 -8001.208,E2 -8001.208} C_VEL
LIN {X 0,Y 459.665,Z 699.005,A -85,B 0,C 180,E1 -8002.973,E2 -8002.973} C_VEL
LIN {X 0,Y 459.597,Z 703.333,A -85,B 0,C 180,E1 -8004.734,E2 -8004.734} C_VEL
LIN {X 0,Y 459.536,Z 706.371,A -85,B 0,C 180,E1 -8006.491,E2 -8006.491} C_VEL
LIN {X 0,Y 459.539,Z 708.19,A -85,B 0,C 180,E1 -8008.246,E2 -8008.246} C_VEL
LIN {X 0,Y 459.527,Z 708.824,A -85,B 0,C 180,E1 -8009.999,E2 -8009.999} C_VEL
LIN {X 0,Y 459.539,Z 708.229,A -85,B 0,C 180,E1 -8011.751,E2 -8011.751} C_VEL
LIN {X 0,Y 459.565,Z 706.449,A -85,B 0,C 180,E1 -8013.506,E2 -8013.506} C_VEL
LIN {X 0,Y 459.602,Z 703.46,A -85,B 0,C 180,E1 -8015.263,E2 -8015.263} C_VEL
LIN {X 0,Y 459.728,Z 699.192,A -85,B 0,C 180,E1 -8017.023,E2 -8017.023} C_VEL
LIN {X 0,Y 459.87,Z 693.527,A -85,B 0,C 180,E1 -8018.789,E2 -8018.789} C_VEL
LIN {X 0,Y 460.2,Z 686.317,A -85,B 0,C 180,E1 -8020.558,E2 -8020.558} C_VEL
LIN {X 0,Y 460.561,Z 678.589,A -85,B 0,C 180,E1 -8022.11,E2 -8022.11} C_VEL
LIN {X 0,Y 461.109,Z 669.27,A -85,B 0,C 180,E1 -8023.663,E2 -8023.663} C_VEL
LIN {X 0,Y 461.679,Z 659.765,A -85,B 0,C 180,E1 -8024.997,E2 -8024.997} C_VEL
LIN {X 0,Y 462.535,Z 647.46,A -85,B 0,C 180,E1 -8026.438,E2 -8026.438} C_VEL
LIN {X 0,Y 463.318,Z 634.884,A -85,B 0,C 180,E1 -8027.659,E2 -8027.659} C_VEL
LIN {X 0,Y 464.247,Z 620.977,A -85,B 0,C 180,E1 -8028.764,E2 -8028.764} C_VEL
LIN {X 0,Y 465.077,Z 607.32,A -85,B 0,C 180,E1 -8029.646,E2 -8029.646} C_VEL
LIN {X 0,Y 465.802,Z 593.484,A -85,B 0,C 180,E1 -8030.36,E2 -8030.36} C_VEL
LIN {X 0,Y 466.418,Z 578.123,A -85,B 0,C 180,E1 -8030.962,E2 -8030.962} C_VEL
LIN {X 0,Y 466.921,Z 562.825,A -85,B 0,C 180,E1 -8031.377,E2 -8031.377} C_VEL
LIN {X 0,Y 469.121,Z 421.244,A -85,B 0,C 180,E1 -8033.769,E2 -8033.769} C_VEL
LIN {X 0,Y 464.469,Z 396.779,A -85,B 0,C 180,E1 -8034.469,E2 -8034.469} C_VEL
LIN {X 0,Y 465.444,Z 378.699,A -85,B 0,C 180,E1 -8037.176,E2 -8037.176} C_VEL
LIN {X 0,Y 462.368,Z 365.116,A -85,B 0,C 180,E1 -8039.484,E2 -8039.484} C_VEL
LIN {X 0,Y 460.525,Z 357.746,A -85,B 0,C 180,E1 -8040.808,E2 -8040.808} C_VEL
LIN {X 0,Y 460.511,Z 357.746,A -85,B 0,C 180,E1 -8043.324,E2 -8043.324} C_VEL
LIN {X 0,Y 460.456,Z 357.755,A -85,B 0,C 180,E1 -8046.529,E2 -8046.529} C_VEL
LIN {X 0,Y 460.5,Z 357.749,A -85,B 0,C 180,E1 -8049.863,E2 -8049.863} C_VEL
LIN {X 0,Y 460.468,Z 357.748,A -85,B 0,C 180,E1 -8052.894,E2 -8052.894} C_VEL
LIN {X 0,Y 460.492,Z 357.748,A -85,B 0,C 180,E1 -8055.83,E2 -8055.83} C_VEL
LIN {X 0,Y 460.502,Z 357.743,A -85,B 0,C 180,E1 -8058.986,E2 -8058.986} C_VEL
LIN {X 0,Y 460.47,Z 357.752,A -85,B 0,C 180,E1 -8062.374,E2 -8062.374} C_VEL
LIN {X 0,Y 460.53,Z 357.742,A -85,B 0,C 180,E1 -8065.623,E2 -8065.623} C_VEL
LIN {X 0,Y 460.524,Z 357.742,A -85,B 0,C 180,E1 -8068.744,E2 -8068.744} C_VEL
LIN {X 0,Y 460.492,Z 357.748,A -85,B 0,C 180,E1 -8071.763,E2 -8071.763} C_VEL
LIN {X 0,Y 460.507,Z 357.744,A -85,B 0,C 180,E1 -8074.703,E2 -8074.703} C_VEL
LIN {X 0,Y 460.492,Z 357.746,A -85,B 0,C 180,E1 -8077.571,E2 -8077.571} C_VEL
LIN {X 0,Y 460.55,Z 357.741,A -85,B 0,C 180,E1 -8080.384,E2 -8080.384} C_VEL
LIN {X 0,Y 460.551,Z 357.745,A -85,B 0,C 180,E1 -8084.057,E2 -8084.057} C_VEL
LIN {X 0,Y 460.594,Z 357.735,A -85,B 0,C 180,E1 -8087.666,E2 -8087.666} C_VEL
LIN {X 0,Y 460.593,Z 357.732,A -85,B 0,C 180,E1 -8091.223,E2 -8091.223} C_VEL
LIN {X 0,Y 460.656,Z 357.73,A -85,B 0,C 180,E1 -8093.87,E2 -8093.87} C_VEL
LIN {X 0,Y 460.74,Z 357.714,A -85,B 0,C 180,E1 -8097.377,E2 -8097.377} C_VEL
LIN {X 0,Y 460.803,Z 357.714,A -85,B 0,C 180,E1 -8100,E2 -8100} C_VEL
LIN {X 0,Y 460.74,Z 357.715,A -85,B 0,C 180,E1 -8102.623,E2 -8102.623} C_VEL
LIN {X 0,Y 460.652,Z 357.731,A -85,B 0,C 180,E1 -8106.131,E2 -8106.131} C_VEL
LIN {X 0,Y 460.588,Z 357.733,A -85,B 0,C 180,E1 -8108.777,E2 -8108.777} C_VEL
LIN {X 0,Y 460.582,Z 357.735,A -85,B 0,C 180,E1 -8112.436,E2 -8112.436} C_VEL
LIN {X 0,Y 460.542,Z 357.746,A -85,B 0,C 180,E1 -8115.979,E2 -8115.979} C_VEL
LIN {X 0,Y 460.551,Z 357.741,A -85,B 0,C 180,E1 -8119.617,E2 -8119.617} C_VEL
LIN {X 0,Y 460.493,Z 357.746,A -85,B 0,C 180,E1 -8122.43,E2 -8122.43} C_VEL
LIN {X 0,Y 460.521,Z 357.747,A -85,B 0,C 180,E1 -8125.794,E2 -8125.794} C_VEL
LIN {X 0,Y 460.506,Z 357.743,A -85,B 0,C 180,E1 -8129.234,E2 -8129.234} C_VEL
LIN {X 0,Y 460.518,Z 357.744,A -85,B 0,C 180,E1 -8132.286,E2 -8132.286} C_VEL
LIN {X 0,Y 460.491,Z 357.747,A -85,B 0,C 180,E1 -8135.448,E2 -8135.448} C_VEL
LIN {X 0,Y 460.481,Z 357.746,A -85,B 0,C 180,E1 -8138.891,E2 -8138.891} C_VEL
LIN {X 0,Y 460.492,Z 357.749,A -85,B 0,C 180,E1 -8141.6,E2 -8141.6} C_VEL
LIN {X 0,Y 460.502,Z 357.744,A -85,B 0,C 180,E1 -8144.591,E2 -8144.591} C_VEL
LIN {X 0,Y 460.471,Z 357.755,A -85,B 0,C 180,E1 -8147.815,E2 -8147.815} C_VEL
LIN {X 0,Y 460.503,Z 357.747,A -85,B 0,C 180,E1 -8150.137,E2 -8150.137} C_VEL
LIN {X 0,Y 460.459,Z 357.752,A -85,B 0,C 180,E1 -8153.471,E2 -8153.471} C_VEL
LIN {X 0,Y 460.514,Z 357.742,A -85,B 0,C 180,E1 -8156.676,E2 -8156.676} C_VEL
LIN {X 0,Y 460.499,Z 357.752,A -85,B 0,C 180,E1 -8159.761,E2 -8159.761} C_VEL
LIN {X 0,Y 460.485,Z 357.745,A -85,B 0,C 180,E1 -8162.752,E2 -8162.752} C_VEL
LIN {X 0,Y 460.514,Z 357.749,A -85,B 0,C 180,E1 -8165.668,E2 -8165.668} C_VEL
LIN {X 0,Y 460.52,Z 357.741,A -85,B 0,C 180,E1 -8168.58,E2 -8168.58} C_VEL
LIN {X 0,Y 460.583,Z 357.736,A -85,B 0,C 180,E1 -8171.312,E2 -8171.312} C_VEL
LIN {X 0,Y 460.605,Z 357.734,A -85,B 0,C 180,E1 -8174.061,E2 -8174.061} C_VEL
LIN {X 0,Y 460.61,Z 357.738,A -85,B 0,C 180,E1 -8177.667,E2 -8177.667} C_VEL
LIN {X 0,Y 460.572,Z 357.736,A -85,B 0,C 180,E1 -8179.194,E2 -8179.194} C_VEL
LIN {X 0,Y 459.907,Z 357.825,A -85,B 0,C 180,E1 -8179.924,E2 -8179.924} C_VEL
LIN {X 0,Y 457.068,Z 358.176,A -85,B 0,C 180,E1 -8181.109,E2 -8181.109} C_VEL
LIN {X 0,Y 454.677,Z 358.472,A -85,B 0,C 180,E1 -8182.066,E2 -8182.066} C_VEL
LIN {X 0,Y 453.663,Z 358.595,A -85,B 0,C 180,E1 -8182.804,E2 -8182.804} C_VEL
LIN {X 0,Y 453.587,Z 358.605,A -85,B 0,C 180,E1 -8183.054,E2 -8183.054} C_VEL
LIN {X 0,Y 453.651,Z 358.597,A -85,B 0,C 180,E1 -8184.668,E2 -8184.668} C_VEL
LIN {X 0,Y 453.69,Z 358.593,A -85,B 0,C 180,E1 -8188.226,E2 -8188.226} C_VEL
LIN {X 0,Y 453.792,Z 358.583,A -85,B 0,C 180,E1 -8190.001,E2 -8190.001} C_VEL
LIN {X 0,Y 453.709,Z 358.589,A -85,B 0,C 180,E1 -8192.665,E2 -8192.665} C_VEL
LIN {X 0,Y 453.642,Z 358.599,A -85,B 0,C 180,E1 -8196.227,E2 -8196.227} C_VEL
LIN {X 0,Y 453.588,Z 358.605,A -85,B 0,C 180,E1 -8198.915,E2 -8198.915} C_VEL
LIN {X 0,Y 453.569,Z 358.607,A -85,B 0,C 180,E1 -8202.53,E2 -8202.53} C_VEL
LIN {X 0,Y 453.508,Z 358.616,A -85,B 0,C 180,E1 -8206.092,E2 -8206.092} C_VEL
LIN {X 0,Y 453.522,Z 358.614,A -85,B 0,C 180,E1 -8209.04,E2 -8209.04} C_VEL
LIN {X 0,Y 453.483,Z 358.622,A -85,B 0,C 180,E1 -8211.837,E2 -8211.837} C_VEL
LIN {X 0,Y 453.475,Z 358.619,A -85,B 0,C 180,E1 -8214.738,E2 -8214.738} C_VEL
LIN {X 0,Y 453.469,Z 358.622,A -85,B 0,C 180,E1 -8217.944,E2 -8217.944} C_VEL
LIN {X 0,Y 453.48,Z 358.618,A -85,B 0,C 180,E1 -8220.76,E2 -8220.76} C_VEL
LIN {X 0,Y 453.481,Z 358.621,A -85,B 0,C 180,E1 -8223.913,E2 -8223.913} C_VEL
LIN {X 0,Y 453.456,Z 358.629,A -85,B 0,C 180,E1 -8227.191,E2 -8227.191} C_VEL
LIN {X 0,Y 453.5,Z 358.62,A -85,B 0,C 180,E1 -8230.609,E2 -8230.609} C_VEL
LIN {X 0,Y 453.493,Z 358.802,A -85,B 0,C 180,E1 -8233.56,E2 -8233.56} C_VEL
LIN {X 0,Y 456.669,Z 372.599,A -85,B 0,C 180,E1 -8236.2,E2 -8236.2} C_VEL
LIN {X 0,Y 459.466,Z 380.313,A -85,B 0,C 180,E1 -8236.499,E2 -8236.499} C_VEL
LIN {X 0,Y 462.765,Z 395.428,A -85,B 0,C 180,E1 -8236.955,E2 -8236.955} C_VEL
LIN {X 0,Y 460.337,Z 538.441,A -85,B 0,C 180,E1 -8239.427,E2 -8239.427} C_VEL
LIN {X 0,Y 459.809,Z 554.122,A -85,B 0,C 180,E1 -8239.878,E2 -8239.878} C_VEL
LIN {X 0,Y 459.147,Z 569.078,A -85,B 0,C 180,E1 -8240.492,E2 -8240.492} C_VEL
LIN {X 0,Y 458.382,Z 583.519,A -85,B 0,C 180,E1 -8241.271,E2 -8241.271} C_VEL
LIN {X 0,Y 457.561,Z 597.783,A -85,B 0,C 180,E1 -8242.245,E2 -8242.245} C_VEL
LIN {X 0,Y 456.768,Z 609.53,A -85,B 0,C 180,E1 -8243.216,E2 -8243.216} C_VEL
LIN {X 0,Y 455.991,Z 621.188,A -85,B 0,C 180,E1 -8244.372,E2 -8244.372} C_VEL
LIN {X 0,Y 455.153,Z 632.417,A -85,B 0,C 180,E1 -8245.695,E2 -8245.695} C_VEL
LIN {X 0,Y 454.392,Z 643.257,A -85,B 0,C 180,E1 -8247.225,E2 -8247.225} C_VEL
LIN {X 0,Y 453.836,Z 652.212,A -85,B 0,C 180,E1 -8248.75,E2 -8248.75} C_VEL
LIN {X 0,Y 453.313,Z 660.778,A -85,B 0,C 180,E1 -8250.512,E2 -8250.512} C_VEL
LIN {X 0,Y 452.929,Z 667.618,A -85,B 0,C 180,E1 -8252.257,E2 -8252.257} C_VEL
LIN {X 0,Y 452.732,Z 672.287,A -85,B 0,C 180,E1 -8253.742,E2 -8253.742} C_VEL
LIN {X 0,Y 452.567,Z 676.033,A -85,B 0,C 180,E1 -8255.21,E2 -8255.21} C_VEL
LIN {X 0,Y 452.382,Z 679.593,A -85,B 0,C 180,E1 -8257.145,E2 -8257.145} C_VEL
LIN {X 0,Y 452.373,Z 681.711,A -85,B 0,C 180,E1 -8259.064,E2 -8259.064} C_VEL
LIN {X 0,Y 452.343,Z 682.461,A -85,B 0,C 180,E1 -8260.957,E2 -8260.957} C_VEL
LIN {X 0,Y 452.324,Z 681.901,A -85,B 0,C 180,E1 -8262.829,E2 -8262.829} C_VEL
LIN {X 0,Y 452.415,Z 680.064,A -85,B 0,C 180,E1 -8264.687,E2 -8264.687} C_VEL
LIN {X 0,Y 452.496,Z 676.956,A -85,B 0,C 180,E1 -8266.527,E2 -8266.527} C_VEL
LIN {X 0,Y 452.742,Z 672.526,A -85,B 0,C 180,E1 -8268.357,E2 -8268.357} C_VEL
LIN {X 0,Y 452.968,Z 666.721,A -85,B 0,C 180,E1 -8270.173,E2 -8270.173} C_VEL
LIN {X 0,Y 453.415,Z 659.364,A -85,B 0,C 180,E1 -8271.981,E2 -8271.981} C_VEL
LIN {X 0,Y 453.924,Z 651.5,A -85,B 0,C 180,E1 -8273.555,E2 -8273.555} C_VEL
LIN {X 0,Y 454.525,Z 642.096,A -85,B 0,C 180,E1 -8275.121,E2 -8275.121} C_VEL
LIN {X 0,Y 455.214,Z 632.53,A -85,B 0,C 180,E1 -8276.459,E2 -8276.459} C_VEL
LIN {X 0,Y 456.044,Z 621.193,A -85,B 0,C 180,E1 -8277.792,E2 -8277.792} C_VEL
LIN {X 0,Y 456.9,Z 609.339,A -85,B 0,C 180,E1 -8278.96,E2 -8278.96} C_VEL
LIN {X 0,Y 457.803,Z 596.634,A -85,B 0,C 180,E1 -8280,E2 -8280} C_VEL
LIN {X 0,Y 458.577,Z 583.582,A -85,B 0,C 180,E1 -8280.878,E2 -8280.878} C_VEL
LIN {X 0,Y 459.366,Z 568.178,A -85,B 0,C 180,E1 -8281.698,E2 -8281.698} C_VEL
LIN {X 0,Y 460.035,Z 552.334,A -85,B 0,C 180,E1 -8282.325,E2 -8282.325} C_VEL
LIN {X 0,Y 460.535,Z 537.513,A -85,B 0,C 180,E1 -8282.733,E2 -8282.733} C_VEL
LIN {X 0,Y 463.229,Z 403.161,A -85,B 0,C 180,E1 -8285.165,E2 -8285.165} C_VEL
LIN {X 0,Y 463.23,Z 394.342,A -85,B 0,C 180,E1 -8285.342,E2 -8285.342} C_VEL
LIN {X 0,Y 459.822,Z 380.111,A -85,B 0,C 180,E1 -8285.849,E2 -8285.849} C_VEL
LIN {X 0,Y 457.326,Z 373.997,A -85,B 0,C 180,E1 -8286.175,E2 -8286.175} C_VEL
LIN {X 0,Y 454.755,Z 363.132,A -85,B 0,C 180,E1 -8288.469,E2 -8288.469} C_VEL
LIN {X 0,Y 453.585,Z 358.614,A -85,B 0,C 180,E1 -8289.475,E2 -8289.475} C_VEL
LIN {X 0,Y 453.569,Z 358.613,A -85,B 0,C 180,E1 -8292.528,E2 -8292.528} C_VEL
LIN {X 0,Y 453.549,Z 358.617,A -85,B 0,C 180,E1 -8296.196,E2 -8296.196} C_VEL
LIN {X 0,Y 453.521,Z 358.618,A -85,B 0,C 180,E1 -8299.039,E2 -8299.039} C_VEL
LIN {X 0,Y 453.481,Z 358.622,A -85,B 0,C 180,E1 -8301.836,E2 -8301.836} C_VEL
LIN {X 0,Y 453.472,Z 358.624,A -85,B 0,C 180,E1 -8304.737,E2 -8304.737} C_VEL
LIN {X 0,Y 453.465,Z 358.627,A -85,B 0,C 180,E1 -8307.942,E2 -8307.942} C_VEL
LIN {X 0,Y 453.46,Z 358.624,A -85,B 0,C 180,E1 -8310.761,E2 -8310.761} C_VEL
LIN {X 0,Y 453.468,Z 358.626,A -85,B 0,C 180,E1 -8313.913,E2 -8313.913} C_VEL
LIN {X 0,Y 453.437,Z 358.626,A -85,B 0,C 180,E1 -8317.191,E2 -8317.191} C_VEL
LIN {X 0,Y 453.469,Z 358.624,A -85,B 0,C 180,E1 -8320.611,E2 -8320.611} C_VEL
LIN {X 0,Y 453.478,Z 358.62,A -85,B 0,C 180,E1 -8324.527,E2 -8324.527} C_VEL
LIN {X 0,Y 453.433,Z 358.63,A -85,B 0,C 180,E1 -8328.071,E2 -8328.071} C_VEL
LIN {X 0,Y 453.426,Z 358.629,A -85,B 0,C 180,E1 -8330.804,E2 -8330.804} C_VEL
LIN {X 0,Y 453.44,Z 358.631,A -85,B 0,C 180,E1 -8333.915,E2 -8333.915} C_VEL
LIN {X 0,Y 453.467,Z 358.63,A -85,B 0,C 180,E1 -8336.815,E2 -8336.815} C_VEL
LIN {X 0,Y 453.464,Z 358.712,A -85,B 0,C 180,E1 -8338.475,E2 -8338.475} C_VEL
LIN {X 0,Y 456.506,Z 370.116,A -85,B 0,C 180,E1 -8340.708,E2 -8340.708} C_VEL
LIN {X 0,Y 458.8,Z 380.969,A -85,B 0,C 180,E1 -8342.68,E2 -8342.68} C_VEL
LIN {X 0,Y 457.826,Z 395.282,A -85,B 0,C 180,E1 -8344.917,E2 -8344.917} C_VEL
LIN {X 0,Y 461.661,Z 414.737,A -85,B 0,C 180,E1 -8345.561,E2 -8345.561} C_VEL
LIN {X 0,Y 463.026,Z 423.572,A -85,B 0,C 180,E1 -8345.823,E2 -8345.823} C_VEL
LIN {X 0,Y 460.747,Z 538.132,A -85,B 0,C 180,E1 -8347.877,E2 -8347.877} C_VEL
LIN {X 0,Y 460.212,Z 564.844,A -85,B 0,C 180,E1 -8348.381,E2 -8348.381} C_VEL
LIN {X 0,Y 459.529,Z 580.593,A -85,B 0,C 180,E1 -8348.855,E2 -8348.855} C_VEL
LIN {X 0,Y 458.791,Z 596.649,A -85,B 0,C 180,E1 -8349.545,E2 -8349.545} C_VEL
LIN {X 0,Y 458.058,Z 609.72,A -85,B 0,C 180,E1 -8350.271,E2 -8350.271} C_VEL
LIN {X 0,Y 457.222,Z 622.817,A -85,B 0,C 180,E1 -8351.167,E2 -8351.167} C_VEL
LIN {X 0,Y 456.352,Z 635.051,A -85,B 0,C 180,E1 -8352.176,E2 -8352.176} C_VEL
LIN {X 0,Y 455.482,Z 647.776,A -85,B 0,C 180,E1 -8353.442,E2 -8353.442} C_VEL
LIN {X 0,Y 454.668,Z 658.918,A -85,B 0,C 180,E1 -8354.764,E2 -8354.764} C_VEL
LIN {X 0,Y 454.095,Z 668.505,A -85,B 0,C 180,E1 -8356.119,E2 -8356.119} C_VEL
LIN {X 0,Y 453.463,Z 677.864,A -85,B 0,C 180,E1 -8357.683,E2 -8357.683} C_VEL
LIN {X 0,Y 453.136,Z 685.749,A -85,B 0,C 180,E1 -8359.273,E2 -8359.273} C_VEL
LIN {X 0,Y 452.782,Z 693.039,A -85,B 0,C 180,E1 -8361.069,E2 -8361.069} C_VEL
LIN {X 0,Y 452.586,Z 698.773,A -85,B 0,C 180,E1 -8362.863,E2 -8362.863} C_VEL
LIN {X 0,Y 452.513,Z 703.113,A -85,B 0,C 180,E1 -8364.652,E2 -8364.652} C_VEL
LIN {X 0,Y 452.433,Z 706.158,A -85,B 0,C 180,E1 -8366.436,E2 -8366.436} C_VEL
LIN {X 0,Y 452.453,Z 707.983,A -85,B 0,C 180,E1 -8368.218,E2 -8368.218} C_VEL
LIN {X 0,Y 452.431,Z 708.618,A -85,B 0,C 180,E1 -8369.999,E2 -8369.999} C_VEL
LIN {X 0,Y 452.453,Z 708.022,A -85,B 0,C 180,E1 -8371.779,E2 -8371.779} C_VEL
LIN {X 0,Y 452.461,Z 706.233,A -85,B 0,C 180,E1 -8373.561,E2 -8373.561} C_VEL
LIN {X 0,Y 452.518,Z 703.231,A -85,B 0,C 180,E1 -8375.345,E2 -8375.345} C_VEL
LIN {X 0,Y 452.646,Z 698.943,A -85,B 0,C 180,E1 -8377.134,E2 -8377.134} C_VEL
LIN {X 0,Y 452.797,Z 693.253,A -85,B 0,C 180,E1 -8378.928,E2 -8378.928} C_VEL
LIN {X 0,Y 453.137,Z 686.011,A -85,B 0,C 180,E1 -8380.725,E2 -8380.725} C_VEL
LIN {X 0,Y 453.527,Z 677.956,A -85,B 0,C 180,E1 -8382.354,E2 -8382.354} C_VEL
LIN {X 0,Y 454.111,Z 668.888,A -85,B 0,C 180,E1 -8383.878,E2 -8383.878} C_VEL
LIN {X 0,Y 454.724,Z 659.355,A -85,B 0,C 180,E1 -8385.231,E2 -8385.231} C_VEL
LIN {X 0,Y 455.554,Z 648.033,A -85,B 0,C 180,E1 -8386.582,E2 -8386.582} C_VEL
LIN {X 0,Y 456.372,Z 635.601,A -85,B 0,C 180,E1 -8387.821,E2 -8387.821} C_VEL
LIN {X 0,Y 457.355,Z 621.911,A -85,B 0,C 180,E1 -8388.941,E2 -8388.941} C_VEL
LIN {X 0,Y 458.219,Z 608.48,A -85,B 0,C 180,E1 -8389.835,E2 -8389.835} C_VEL
LIN {X 0,Y 459.025,Z 593.756,A -85,B 0,C 180,E1 -8390.617,E2 -8390.617} C_VEL
LIN {X 0,Y 459.677,Z 577.913,A -85,B 0,C 180,E1 -8391.25,E2 -8391.25} C_VEL
LIN {X 0,Y 460.23,Z 562.395,A -85,B 0,C 180,E1 -8391.674,E2 -8391.674} C_VEL
LIN {X 0,Y 462.571,Z 422.141,A -85,B 0,C 180,E1 -8394.087,E2 -8394.087} C_VEL
LIN {X 0,Y 457.677,Z 396.699,A -85,B 0,C 180,E1 -8394.824,E2 -8394.824} C_VEL
LIN {X 0,Y 458.634,Z 380.546,A -85,B 0,C 180,E1 -8397.28,E2 -8397.28} C_VEL
LIN {X 0,Y 455.622,Z 367.209,A -85,B 0,C 180,E1 -8399.576,E2 -8399.576} C_VEL
LIN {X 0,Y 453.504,Z 358.621,A -85,B 0,C 180,E1 -8401.124,E2 -8401.124} C_VEL
LIN {X 0,Y 453.459,Z 358.626,A -85,B 0,C 180,E1 -8403.912,E2 -8403.912} C_VEL
LIN {X 0,Y 453.429,Z 358.627,A -85,B 0,C 180,E1 -8407.19,E2 -8407.19} C_VEL
LIN {X 0,Y 453.46,Z 358.623,A -85,B 0,C 180,E1 -8410.61,E2 -8410.61} C_VEL
LIN {X 0,Y 453.447,Z 358.63,A -85,B 0,C 180,E1 -8414.221,E2 -8414.221} C_VEL
LIN {X 0,Y 453.413,Z 358.626,A -85,B 0,C 180,E1 -8416.999,E2 -8416.999} C_VEL
LIN {X 0,Y 453.458,Z 358.621,A -85,B 0,C 180,E1 -8419.412,E2 -8419.412} C_VEL
LIN {X 0,Y 453.423,Z 358.626,A -85,B 0,C 180,E1 -8422.808,E2 -8422.808} C_VEL
LIN {X 0,Y 453.461,Z 358.628,A -85,B 0,C 180,E1 -8426.086,E2 -8426.086} C_VEL
LIN {X 0,Y 453.46,Z 358.62,A -85,B 0,C 180,E1 -8429.239,E2 -8429.239} C_VEL
LIN {X 0,Y 453.459,Z 358.626,A -85,B 0,C 180,E1 -8432.293,E2 -8432.293} C_VEL
LIN {X 0,Y 453.454,Z 358.621,A -85,B 0,C 180,E1 -8435.262,E2 -8435.262} C_VEL
LIN {X 0,Y 453.465,Z 358.624,A -85,B 0,C 180,E1 -8438.415,E2 -8438.415} C_VEL
LIN {X 0,Y 453.508,Z 358.614,A -85,B 0,C 180,E1 -8441.008,E2 -8441.008} C_VEL
LIN {X 0,Y 453.503,Z 358.616,A -85,B 0,C 180,E1 -8444.725,E2 -8444.725} C_VEL
LIN {X 0,Y 453.542,Z 358.614,A -85,B 0,C 180,E1 -8448.379,E2 -8448.379} C_VEL
LIN {X 0,Y 453.561,Z 358.608,A -85,B 0,C 180,E1 -8451.086,E2 -8451.086} C_VEL
LIN {X 0,Y 453.623,Z 358.605,A -85,B 0,C 180,E1 -8453.774,E2 -8453.774} C_VEL
LIN {X 0,Y 453.687,Z 358.593,A -85,B 0,C 180,E1 -8457.337,E2 -8457.337} C_VEL
LIN {X 0,Y 453.772,Z 358.59,A -85,B 0,C 180,E1 -8460,E2 -8460} C_VEL
LIN {X 0,Y 453.686,Z 358.593,A -85,B 0,C 180,E1 -8462.664,E2 -8462.664} C_VEL
LIN {X 0,Y 453.62,Z 358.605,A -85,B 0,C 180,E1 -8466.226,E2 -8466.226} C_VEL
LIN {X 0,Y 453.554,Z 358.609,A -85,B 0,C 180,E1 -8468.914,E2 -8468.914} C_VEL
LIN {X 0,Y 453.55,Z 358.611,A -85,B 0,C 180,E1 -8472.53,E2 -8472.53} C_VEL
LIN {X 0,Y 453.488,Z 358.623,A -85,B 0,C 180,E1 -8476.092,E2 -8476.092} C_VEL
LIN {X 0,Y 453.503,Z 358.615,A -85,B 0,C 180,E1 -8479.04,E2 -8479.04} C_VEL
LIN {X 0,Y 453.462,Z 358.627,A -85,B 0,C 180,E1 -8481.837,E2 -8481.837} C_VEL
LIN {X 0,Y 453.456,Z 358.621,A -85,B 0,C 180,E1 -8484.738,E2 -8484.738} C_VEL
LIN {X 0,Y 453.449,Z 358.629,A -85,B 0,C 180,E1 -8487.944,E2 -8487.944} C_VEL
LIN {X 0,Y 453.462,Z 358.62,A -85,B 0,C 180,E1 -8490.761,E2 -8490.761} C_VEL
LIN {X 0,Y 453.456,Z 358.629,A -85,B 0,C 180,E1 -8493.915,E2 -8493.915} C_VEL
LIN {X 0,Y 453.425,Z 358.626,A -85,B 0,C 180,E1 -8497.193,E2 -8497.193} C_VEL
LIN {X 0,Y 453.46,Z 358.621,A -85,B 0,C 180,E1 -8500.613,E2 -8500.613} C_VEL
LIN {X 0,Y 453.472,Z 358.62,A -85,B 0,C 180,E1 -8504.53,E2 -8504.53} C_VEL
LIN {X 0,Y 453.431,Z 358.629,A -85,B 0,C 180,E1 -8508.072,E2 -8508.072} C_VEL
LIN {X 0,Y 453.432,Z 358.624,A -85,B 0,C 180,E1 -8510.804,E2 -8510.804} C_VEL
LIN {X 0,Y 453.441,Z 358.629,A -85,B 0,C 180,E1 -8513.918,E2 -8513.918} C_VEL
LIN {X 0,Y 453.473,Z 358.62,A -85,B 0,C 180,E1 -8517.152,E2 -8517.152} C_VEL
LIN {X 0,Y 453.457,Z 358.623,A -85,B 0,C 180,E1 -8520.269,E2 -8520.269} C_VEL
LIN {X 0,Y 453.436,Z 358.626,A -85,B 0,C 180,E1 -8523.291,E2 -8523.291} C_VEL
LIN {X 0,Y 453.49,Z 358.619,A -85,B 0,C 180,E1 -8526.24,E2 -8526.24} C_VEL
LIN {X 0,Y 453.48,Z 358.619,A -85,B 0,C 180,E1 -8529.119,E2 -8529.119} C_VEL
LIN {X 0,Y 453.497,Z 358.621,A -85,B 0,C 180,E1 -8531.946,E2 -8531.946} C_VEL
LIN {X 0,Y 453.537,Z 358.611,A -85,B 0,C 180,E1 -8534.728,E2 -8534.728} C_VEL
LIN {X 0,Y 453.559,Z 358.609,A -85,B 0,C 180,E1 -8538.38,E2 -8538.38} C_VEL
LIN {X 0,Y 453.578,Z 358.607,A -85,B 0,C 180,E1 -8541.088,E2 -8541.088} C_VEL
LIN {X 0,Y 453.587,Z 358.605,A -85,B 0,C 180,E1 -8543.054,E2 -8543.054} C_VEL
LIN {X 0,Y 452.906,Z 358.696,A -85,B 0,C 180,E1 -8543.795,E2 -8543.795} C_VEL
LIN {X 0,Y 449.958,Z 359.057,A -85,B 0,C 180,E1 -8544.997,E2 -8544.997} C_VEL
LIN {X 0,Y 447.529,Z 359.363,A -85,B 0,C 180,E1 -8545.967,E2 -8545.967} C_VEL
LIN {X 0,Y 446.585,Z 359.477,A -85,B 0,C 180,E1 -8546.718,E2 -8546.718} C_VEL
LIN {X 0,Y 446.562,Z 359.48,A -85,B 0,C 180,E1 -8546.972,E2 -8546.972} C_VEL
LIN {X 0,Y 446.741,Z 359.461,A -85,B 0,C 180,E1 -8550.001,E2 -8550.001} C_VEL
LIN {X 0,Y 446.658,Z 359.468,A -85,B 0,C 180,E1 -8552.707,E2 -8552.707} C_VEL
LIN {X 0,Y 446.612,Z 359.474,A -85,B 0,C 180,E1 -8556.325,E2 -8556.325} C_VEL
LIN {X 0,Y 446.535,Z 359.485,A -85,B 0,C 180,E1 -8559.057,E2 -8559.057} C_VEL
LIN {X 0,Y 446.527,Z 359.484,A -85,B 0,C 180,E1 -8562.731,E2 -8562.731} C_VEL
LIN {X 0,Y 446.459,Z 359.494,A -85,B 0,C 180,E1 -8566.21,E2 -8566.21} C_VEL
LIN {X 0,Y 446.474,Z 359.495,A -85,B 0,C 180,E1 -8569.304,E2 -8569.304} C_VEL
LIN {X 0,Y 446.424,Z 359.498,A -85,B 0,C 180,E1 -8572.2,E2 -8572.2} C_VEL
LIN {X 0,Y 446.427,Z 359.499,A -85,B 0,C 180,E1 -8575.155,E2 -8575.155} C_VEL
LIN {X 0,Y 446.443,Z 359.496,A -85,B 0,C 180,E1 -8578.183,E2 -8578.183} C_VEL
LIN {X 0,Y 446.421,Z 359.502,A -85,B 0,C 180,E1 -8581.301,E2 -8581.301} C_VEL
LIN {X 0,Y 446.434,Z 359.496,A -85,B 0,C 180,E1 -8584.524,E2 -8584.524} C_VEL
LIN {X 0,Y 446.417,Z 359.502,A -85,B 0,C 180,E1 -8588.079,E2 -8588.079} C_VEL
LIN {X 0,Y 446.425,Z 359.505,A -85,B 0,C 180,E1 -8591.393,E2 -8591.393} C_VEL
LIN {X 0,Y 446.448,Z 359.68,A -85,B 0,C 180,E1 -8593.252,E2 -8593.252} C_VEL
LIN {X 0,Y 449.409,Z 372.578,A -85,B 0,C 180,E1 -8595.793,E2 -8595.793} C_VEL
LIN {X 0,Y 453.233,Z 382.705,A -85,B 0,C 180,E1 -8596.203,E2 -8596.203} C_VEL
LIN {X 0,Y 456.176,Z 396.034,A -85,B 0,C 180,E1 -8596.615,E2 -8596.615} C_VEL
LIN {X 0,Y 453.653,Z 538.739,A -85,B 0,C 180,E1 -8599.133,E2 -8599.133} C_VEL
LIN {X 0,Y 453.1,Z 554.257,A -85,B 0,C 180,E1 -8599.587,E2 -8599.587} C_VEL
LIN {X 0,Y 452.405,Z 569.426,A -85,B 0,C 180,E1 -8600.22,E2 -8600.22} C_VEL
LIN {X 0,Y 451.635,Z 583.298,A -85,B 0,C 180,E1 -8600.975,E2 -8600.975} C_VEL
LIN {X 0,Y 450.776,Z 597.92,A -85,B 0,C 180,E1 -8601.987,E2 -8601.987} C_VEL
LIN {X 0,Y 449.826,Z 610.707,A -85,B 0,C 180,E1 -8603.067,E2 -8603.067} C_VEL
LIN {X 0,Y 448.931,Z 623.253,A -85,B 0,C 180,E1 -8604.355,E2 -8604.355} C_VEL
LIN {X 0,Y 448.164,Z 633.693,A -85,B 0,C 180,E1 -8605.629,E2 -8605.629} C_VEL
LIN {X 0,Y 447.381,Z 644.339,A -85,B 0,C 180,E1 -8607.182,E2 -8607.182} C_VEL
LIN {X 0,Y 446.772,Z 653.17,A -85,B 0,C 180,E1 -8608.727,E2 -8608.727} C_VEL
LIN {X 0,Y 446.267,Z 661.015,A -85,B 0,C 180,E1 -8610.382,E2 -8610.382} C_VEL
LIN {X 0,Y 445.917,Z 667.153,A -85,B 0,C 180,E1 -8611.96,E2 -8611.96} C_VEL
LIN {X 0,Y 445.655,Z 672.893,A -85,B 0,C 180,E1 -8613.796,E2 -8613.796} C_VEL
LIN {X 0,Y 445.474,Z 676.534,A -85,B 0,C 180,E1 -8615.286,E2 -8615.286} C_VEL
LIN {X 0,Y 445.327,Z 679.25,A -85,B 0,C 180,E1 -8616.762,E2 -8616.762} C_VEL
LIN {X 0,Y 445.271,Z 681.615,A -85,B 0,C 180,E1 -8618.714,E2 -8618.714} C_VEL
LIN {X 0,Y 445.246,Z 682.603,A -85,B 0,C 180,E1 -8620.641,E2 -8620.641} C_VEL
LIN {X 0,Y 445.223,Z 682.275,A -85,B 0,C 180,E1 -8622.547,E2 -8622.547} C_VEL
LIN {X 0,Y 445.314,Z 680.665,A -85,B 0,C 180,E1 -8624.437,E2 -8624.437} C_VEL
LIN {X 0,Y 445.401,Z 677.783,A -85,B 0,C 180,E1 -8626.309,E2 -8626.309} C_VEL
LIN {X 0,Y 445.644,Z 673.578,A -85,B 0,C 180,E1 -8628.169,E2 -8628.169} C_VEL
LIN {X 0,Y 445.876,Z 668.013,A -85,B 0,C 180,E1 -8630.015,E2 -8630.015} C_VEL
LIN {X 0,Y 446.374,Z 660.91,A -85,B 0,C 180,E1 -8631.853,E2 -8631.853} C_VEL
LIN {X 0,Y 446.856,Z 653.337,A -85,B 0,C 180,E1 -8633.452,E2 -8633.452} C_VEL
LIN {X 0,Y 447.488,Z 644.242,A -85,B 0,C 180,E1 -8635.044,E2 -8635.044} C_VEL
LIN {X 0,Y 448.312,Z 633.291,A -85,B 0,C 180,E1 -8636.63,E2 -8636.63} C_VEL
LIN {X 0,Y 449.18,Z 622.065,A -85,B 0,C 180,E1 -8637.982,E2 -8637.982} C_VEL
LIN {X 0,Y 450.123,Z 609.67,A -85,B 0,C 180,E1 -8639.226,E2 -8639.226} C_VEL
LIN {X 0,Y 451.115,Z 596.266,A -85,B 0,C 180,E1 -8640.334,E2 -8640.334} C_VEL
LIN {X 0,Y 451.965,Z 583.11,A -85,B 0,C 180,E1 -8641.225,E2 -8641.225} C_VEL
LIN {X 0,Y 452.739,Z 568.702,A -85,B 0,C 180,E1 -8642.001,E2 -8642.001} C_VEL
LIN {X 0,Y 453.429,Z 553.07,A -85,B 0,C 180,E1 -8642.637,E2 -8642.637} C_VEL
LIN {X 0,Y 454.001,Z 537.284,A -85,B 0,C 180,E1 -8643.078,E2 -8643.078} C_VEL
LIN {X 0,Y 456.901,Z 402.077,A -85,B 0,C 180,E1 -8645.584,E2 -8645.584} C_VEL
LIN {X 0,Y 456.865,Z 395.5,A -85,B 0,C 180,E1 -8645.725,E2 -8645.725} C_VEL
LIN {X 0,Y 454,Z 383.261,A -85,B 0,C 180,E1 -8646.178,E2 -8646.178} C_VEL
LIN {X 0,Y 450.244,Z 374.441,A -85,B 0,C 180,E1 -8646.643,E2 -8646.643} C_VEL
LIN {X 0,Y 447.571,Z 363.48,A -85,B 0,C 180,E1 -8649.034,E2 -8649.034} C_VEL
LIN {X 0,Y 446.524,Z 359.492,A -85,B 0,C 180,E1 -8649.97,E2 -8649.97} C_VEL
LIN {X 0,Y 446.527,Z 359.489,A -85,B 0,C 180,E1 -8652.729,E2 -8652.729} C_VEL
LIN {X 0,Y 446.501,Z 359.496,A -85,B 0,C 180,E1 -8656.227,E2 -8656.227} C_VEL
LIN {X 0,Y 446.473,Z 359.495,A -85,B 0,C 180,E1 -8659.303,E2 -8659.303} C_VEL
LIN {X 0,Y 446.423,Z 359.505,A -85,B 0,C 180,E1 -8662.199,E2 -8662.199} C_VEL
LIN {X 0,Y 446.424,Z 359.499,A -85,B 0,C 180,E1 -8665.154,E2 -8665.154} C_VEL
LIN {X 0,Y 446.42,Z 359.504,A -85,B 0,C 180,E1 -8668.183,E2 -8668.183} C_VEL
LIN {X 0,Y 446.411,Z 359.5,A -85,B 0,C 180,E1 -8671.301,E2 -8671.301} C_VEL
LIN {X 0,Y 446.423,Z 359.503,A -85,B 0,C 180,E1 -8674.523,E2 -8674.523} C_VEL
LIN {X 0,Y 446.398,Z 359.507,A -85,B 0,C 180,E1 -8678.075,E2 -8678.075} C_VEL
LIN {X 0,Y 446.398,Z 359.504,A -85,B 0,C 180,E1 -8681.394,E2 -8681.394} C_VEL
LIN {X 0,Y 446.42,Z 359.498,A -85,B 0,C 180,E1 -8685.108,E2 -8685.108} C_VEL
LIN {X 0,Y 446.398,Z 359.503,A -85,B 0,C 180,E1 -8688.604,E2 -8688.604} C_VEL
LIN {X 0,Y 446.39,Z 359.508,A -85,B 0,C 180,E1 -8692.118,E2 -8692.118} C_VEL
LIN {X 0,Y 446.413,Z 359.507,A -85,B 0,C 180,E1 -8695.474,E2 -8695.474} C_VEL
LIN {X 0,Y 446.411,Z 359.61,A -85,B 0,C 180,E1 -8697.999,E2 -8697.999} C_VEL
LIN {X 0,Y 449.766,Z 372.042,A -85,B 0,C 180,E1 -8700.513,E2 -8700.513} C_VEL
LIN {X 0,Y 451.985,Z 382.218,A -85,B 0,C 180,E1 -8702.412,E2 -8702.412} C_VEL
LIN {X 0,Y 451.699,Z 388.466,A -85,B 0,C 180,E1 -8703.427,E2 -8703.427} C_VEL
LIN {X 0,Y 451.226,Z 395.276,A -85,B 0,C 180,E1 -8704.471,E2 -8704.471} C_VEL
LIN {X 0,Y 455.205,Z 415.207,A -85,B 0,C 180,E1 -8705.161,E2 -8705.161} C_VEL
LIN {X 0,Y 456.672,Z 424.467,A -85,B 0,C 180,E1 -8705.447,E2 -8705.447} C_VEL
LIN {X 0,Y 454.137,Z 541.568,A -85,B 0,C 180,E1 -8707.598,E2 -8707.598} C_VEL
LIN {X 0,Y 453.622,Z 564.698,A -85,B 0,C 180,E1 -8708.051,E2 -8708.051} C_VEL
LIN {X 0,Y 452.926,Z 580.413,A -85,B 0,C 180,E1 -8708.533,E2 -8708.533} C_VEL
LIN {X 0,Y 452.119,Z 596.382,A -85,B 0,C 180,E1 -8709.229,E2 -8709.229} C_VEL
LIN {X 0,Y 451.336,Z 609.43,A -85,B 0,C 180,E1 -8709.965,E2 -8709.965} C_VEL
LIN {X 0,Y 450.429,Z 622.517,A -85,B 0,C 180,E1 -8710.872,E2 -8710.872} C_VEL
LIN {X 0,Y 449.429,Z 635.956,A -85,B 0,C 180,E1 -8712.009,E2 -8712.009} C_VEL
LIN {X 0,Y 448.554,Z 647.951,A -85,B 0,C 180,E1 -8713.232,E2 -8713.232} C_VEL
LIN {X 0,Y 447.74,Z 658.637,A -85,B 0,C 180,E1 -8714.522,E2 -8714.522} C_VEL
LIN {X 0,Y 447.117,Z 668.238,A -85,B 0,C 180,E1 -8715.898,E2 -8715.898} C_VEL
LIN {X 0,Y 446.425,Z 677.335,A -85,B 0,C 180,E1 -8717.436,E2 -8717.436} C_VEL
LIN {X 0,Y 446.1,Z 685.503,A -85,B 0,C 180,E1 -8719.101,E2 -8719.101} C_VEL
LIN {X 0,Y 445.699,Z 692.806,A -85,B 0,C 180,E1 -8720.926,E2 -8720.926} C_VEL
LIN {X 0,Y 445.506,Z 698.552,A -85,B 0,C 180,E1 -8722.749,E2 -8722.749} C_VEL
LIN {X 0,Y 445.411,Z 702.899,A -85,B 0,C 180,E1 -8724.566,E2 -8724.566} C_VEL
LIN {X 0,Y 445.333,Z 705.95,A -85,B 0,C 180,E1 -8726.379,E2 -8726.379} C_VEL
LIN {X 0,Y 445.371,Z 707.777,A -85,B 0,C 180,E1 -8728.19,E2 -8728.19} C_VEL
LIN {X 0,Y 445.339,Z 708.412,A -85,B 0,C 180,E1 -8729.999,E2 -8729.999} C_VEL
LIN {X 0,Y 445.371,Z 707.812,A -85,B 0,C 180,E1 -8731.807,E2 -8731.807} C_VEL
LIN {X 0,Y 445.358,Z 706.012,A -85,B 0,C 180,E1 -8733.618,E2 -8733.618} C_VEL
LIN {X 0,Y 445.418,Z 702.994,A -85,B 0,C 180,E1 -8735.431,E2 -8735.431} C_VEL
LIN {X 0,Y 445.569,Z 698.687,A -85,B 0,C 180,E1 -8737.248,E2 -8737.248} C_VEL
LIN {X 0,Y 445.71,Z 692.971,A -85,B 0,C 180,E1 -8739.071,E2 -8739.071} C_VEL
LIN {X 0,Y 446.105,Z 685.696,A -85,B 0,C 180,E1 -8740.896,E2 -8740.896} C_VEL
LIN {X 0,Y 446.507,Z 677.269,A -85,B 0,C 180,E1 -8742.611,E2 -8742.611} C_VEL
LIN {X 0,Y 447.12,Z 668.48,A -85,B 0,C 180,E1 -8744.1,E2 -8744.1} C_VEL
LIN {X 0,Y 447.788,Z 658.902,A -85,B 0,C 180,E1 -8745.473,E2 -8745.473} C_VEL
LIN {X 0,Y 448.644,Z 647.947,A -85,B 0,C 180,E1 -8746.795,E2 -8746.795} C_VEL
LIN {X 0,Y 449.502,Z 635.006,A -85,B 0,C 180,E1 -8748.103,E2 -8748.103} C_VEL
LIN {X 0,Y 450.572,Z 621.208,A -85,B 0,C 180,E1 -8749.237,E2 -8749.237} C_VEL
LIN {X 0,Y 451.443,Z 607.684,A -85,B 0,C 180,E1 -8750.146,E2 -8750.146} C_VEL
LIN {X 0,Y 452.3,Z 592.776,A -85,B 0,C 180,E1 -8750.938,E2 -8750.938} C_VEL
LIN {X 0,Y 452.967,Z 577.663,A -85,B 0,C 180,E1 -8751.545,E2 -8751.545} C_VEL
LIN {X 0,Y 453.563,Z 561.885,A -85,B 0,C 180,E1 -8751.98,E2 -8751.98} C_VEL
LIN {X 0,Y 456.051,Z 424.471,A -85,B 0,C 180,E1 -8754.388,E2 -8754.388} C_VEL
LIN {X 0,Y 454.687,Z 416.248,A -85,B 0,C 180,E1 -8754.614,E2 -8754.614} C_VEL
LIN {X 0,Y 450.885,Z 396.478,A -85,B 0,C 180,E1 -8755.213,E2 -8755.213} C_VEL
LIN {X 0,Y 451.821,Z 382.68,A -85,B 0,C 180,E1 -8757.334,E2 -8757.334} C_VEL
LIN {X 0,Y 449.087,Z 370.055,A -85,B 0,C 180,E1 -8759.533,E2 -8759.533} C_VEL
LIN {X 0,Y 446.419,Z 359.504,A -85,B 0,C 180,E1 -8761.473,E2 -8761.473} C_VEL
LIN {X 0,Y 446.413,Z 359.503,A -85,B 0,C 180,E1 -8764.522,E2 -8764.522} C_VEL
LIN {X 0,Y 446.39,Z 359.508,A -85,B 0,C 180,E1 -8768.075,E2 -8768.075} C_VEL
LIN {X 0,Y 446.396,Z 359.501,A -85,B 0,C 180,E1 -8771.392,E2 -8771.392} C_VEL
LIN {X 0,Y 446.41,Z 359.499,A -85,B 0,C 180,E1 -8774.891,E2 -8774.891} C_VEL
LIN {X 0,Y 446.372,Z 359.506,A -85,B 0,C 180,E1 -8777.729,E2 -8777.729} C_VEL
LIN {X 0,Y 446.386,Z 359.502,A -85,B 0,C 180,E1 -8780.967,E2 -8780.967} C_VEL
LIN {X 0,Y 446.399,Z 359.505,A -85,B 0,C 180,E1 -8784.372,E2 -8784.372} C_VEL
LIN {X 0,Y 446.408,Z 359.501,A -85,B 0,C 180,E1 -8787.637,E2 -8787.637} C_VEL
LIN {X 0,Y 446.407,Z 359.5,A -85,B 0,C 180,E1 -8790.788,E2 -8790.788} C_VEL
LIN {X 0,Y 446.42,Z 359.502,A -85,B 0,C 180,E1 -8793.845,E2 -8793.845} C_VEL
LIN {X 0,Y 446.407,Z 359.5,A -85,B 0,C 180,E1 -8796.822,E2 -8796.822} C_VEL
LIN {X 0,Y 446.427,Z 359.5,A -85,B 0,C 180,E1 -8799.737,E2 -8799.737} C_VEL
LIN {X 0,Y 446.42,Z 359.499,A -85,B 0,C 180,E1 -8802.596,E2 -8802.596} C_VEL
LIN {X 0,Y 446.442,Z 359.496,A -85,B 0,C 180,E1 -8805.412,E2 -8805.412} C_VEL
LIN {X 0,Y 446.501,Z 359.493,A -85,B 0,C 180,E1 -8808.193,E2 -8808.193} C_VEL
LIN {X 0,Y 446.51,Z 359.486,A -85,B 0,C 180,E1 -8810.944,E2 -8810.944} C_VEL
LIN {X 0,Y 446.593,Z 359.479,A -85,B 0,C 180,E1 -8813.676,E2 -8813.676} C_VEL
LIN {X 0,Y 446.636,Z 359.471,A -85,B 0,C 180,E1 -8817.295,E2 -8817.295} C_VEL
LIN {X 0,Y 446.721,Z 359.468,A -85,B 0,C 180,E1 -8820,E2 -8820} C_VEL
LIN {X 0,Y 446.636,Z 359.471,A -85,B 0,C 180,E1 -8822.706,E2 -8822.706} C_VEL
LIN {X 0,Y 446.59,Z 359.48,A -85,B 0,C 180,E1 -8826.325,E2 -8826.325} C_VEL
LIN {X 0,Y 446.502,Z 359.487,A -85,B 0,C 180,E1 -8829.056,E2 -8829.056} C_VEL
LIN {X 0,Y 446.507,Z 359.487,A -85,B 0,C 180,E1 -8832.73,E2 -8832.73} C_VEL
LIN {X 0,Y 446.439,Z 359.499,A -85,B 0,C 180,E1 -8836.21,E2 -8836.21} C_VEL
LIN {X 0,Y 446.454,Z 359.494,A -85,B 0,C 180,E1 -8839.304,E2 -8839.304} C_VEL
LIN {X 0,Y 446.403,Z 359.504,A -85,B 0,C 180,E1 -8842.201,E2 -8842.201} C_VEL
LIN {X 0,Y 446.408,Z 359.499,A -85,B 0,C 180,E1 -8845.156,E2 -8845.156} C_VEL
LIN {X 0,Y 446.404,Z 359.504,A -85,B 0,C 180,E1 -8848.185,E2 -8848.185} C_VEL
LIN {X 0,Y 446.403,Z 359.501,A -85,B 0,C 180,E1 -8851.302,E2 -8851.302} C_VEL
LIN {X 0,Y 446.41,Z 359.5,A -85,B 0,C 180,E1 -8854.525,E2 -8854.525} C_VEL
LIN {X 0,Y 446.387,Z 359.507,A -85,B 0,C 180,E1 -8858.078,E2 -8858.078} C_VEL
LIN {X 0,Y 446.39,Z 359.504,A -85,B 0,C 180,E1 -8861.396,E2 -8861.396} C_VEL
LIN {X 0,Y 446.413,Z 359.499,A -85,B 0,C 180,E1 -8865.109,E2 -8865.109} C_VEL
LIN {X 0,Y 446.394,Z 359.501,A -85,B 0,C 180,E1 -8868.607,E2 -8868.607} C_VEL
LIN {X 0,Y 446.393,Z 359.507,A -85,B 0,C 180,E1 -8871.925,E2 -8871.925} C_VEL
LIN {X 0,Y 446.416,Z 359.502,A -85,B 0,C 180,E1 -8875.478,E2 -8875.478} C_VEL
LIN {X 0,Y 446.41,Z 359.499,A -85,B 0,C 180,E1 -8878.701,E2 -8878.701} C_VEL
LIN {X 0,Y 446.42,Z 359.505,A -85,B 0,C 180,E1 -8881.838,E2 -8881.838} C_VEL
LIN {X 0,Y 446.417,Z 359.498,A -85,B 0,C 180,E1 -8884.847,E2 -8884.847} C_VEL
LIN {X 0,Y 446.447,Z 359.496,A -85,B 0,C 180,E1 -8888.247,E2 -8888.247} C_VEL
LIN {X 0,Y 446.448,Z 359.501,A -85,B 0,C 180,E1 -8891.65,E2 -8891.65} C_VEL
LIN {X 0,Y 446.506,Z 359.487,A -85,B 0,C 180,E1 -8894.481,E2 -8894.481} C_VEL
LIN {X 0,Y 446.518,Z 359.487,A -85,B 0,C 180,E1 -8898.195,E2 -8898.195} C_VEL
LIN {X 0,Y 446.527,Z 359.485,A -85,B 0,C 180,E1 -8900.946,E2 -8900.946} C_VEL
LIN {X 0,Y 446.608,Z 359.482,A -85,B 0,C 180,E1 -8903.677,E2 -8903.677} C_VEL
LIN {X 0,Y 446.562,Z 359.48,A -85,B 0,C 180,E1 -8906.972,E2 -8906.972} C_VEL
LIN {X 0,Y 446.347,Z 359.512,A -85,B 0,C 180,E1 -8907.476,E2 -8907.476} C_VEL
LIN {X 0,Y 445.044,Z 359.673,A -85,B 0,C 180,E1 -8908.218,E2 -8908.218} C_VEL
LIN {X 0,Y 440.623,Z 360.224,A -85,B 0,C 180,E1 -8909.934,E2 -8909.934} C_VEL
LIN {X 0,Y 439.571,Z 360.352,A -85,B 0,C 180,E1 -8910.698,E2 -8910.698} C_VEL
LIN {X 0,Y 439.504,Z 360.359,A -85,B 0,C 180,E1 -8910.957,E2 -8910.957} C_VEL
LIN {X 0,Y 439.61,Z 360.346,A -85,B 0,C 180,E1 -8912.75,E2 -8912.75} C_VEL
LIN {X 0,Y 439.565,Z 360.352,A -85,B 0,C 180,E1 -8916.427,E2 -8916.427} C_VEL
LIN {X 0,Y 439.499,Z 360.362,A -85,B 0,C 180,E1 -8919.203,E2 -8919.203} C_VEL
LIN {X 0,Y 439.47,Z 360.364,A -85,B 0,C 180,E1 -8922.939,E2 -8922.939} C_VEL
LIN {X 0,Y 439.407,Z 360.371,A -85,B 0,C 180,E1 -8926.329,E2 -8926.329} C_VEL
LIN {X 0,Y 439.408,Z 360.378,A -85,B 0,C 180,E1 -8929.627,E2 -8929.627} C_VEL
LIN {X 0,Y 439.369,Z 360.376,A -85,B 0,C 180,E1 -8932.576,E2 -8932.576} C_VEL
LIN {X 0,Y 439.373,Z 360.383,A -85,B 0,C 180,E1 -8935.588,E2 -8935.588} C_VEL
LIN {X 0,Y 439.396,Z 360.372,A -85,B 0,C 180,E1 -8938.676,E2 -8938.676} C_VEL
LIN {X 0,Y 439.376,Z 360.377,A -85,B 0,C 180,E1 -8942.031,E2 -8942.031} C_VEL
LIN {X 0,Y 439.399,Z 360.378,A -85,B 0,C 180,E1 -8945.34,E2 -8945.34} C_VEL
LIN {X 0,Y 439.369,Z 360.38,A -85,B 0,C 180,E1 -8948.598,E2 -8948.598} C_VEL
LIN {X 0,Y 439.388,Z 360.381,A -85,B 0,C 180,E1 -8951.256,E2 -8951.256} C_VEL
LIN {X 0,Y 439.42,Z 360.578,A -85,B 0,C 180,E1 -8952.941,E2 -8952.941} C_VEL
LIN {X 0,Y 442.227,Z 372.708,A -85,B 0,C 180,E1 -8955.377,E2 -8955.377} C_VEL
LIN {X 0,Y 446.909,Z 384.761,A -85,B 0,C 180,E1 -8955.889,E2 -8955.889} C_VEL
LIN {X 0,Y 449.667,Z 397.203,A -85,B 0,C 180,E1 -8956.283,E2 -8956.283} C_VEL
LIN {X 0,Y 446.97,Z 538.881,A -85,B 0,C 180,E1 -8958.832,E2 -8958.832} C_VEL
LIN {X 0,Y 446.383,Z 554.523,A -85,B 0,C 180,E1 -8959.297,E2 -8959.297} C_VEL
LIN {X 0,Y 445.641,Z 570.045,A -85,B 0,C 180,E1 -8959.958,E2 -8959.958} C_VEL
LIN {X 0,Y 444.827,Z 583.922,A -85,B 0,C 180,E1 -8960.731,E2 -8960.731} C_VEL
LIN {X 0,Y 443.962,Z 598.13,A -85,B 0,C 180,E1 -8961.73,E2 -8961.73} C_VEL
LIN {X 0,Y 443.078,Z 610.1,A -85,B 0,C 180,E1 -8962.749,E2 -8962.749} C_VEL
LIN {X 0,Y 442.196,Z 622.134,A -85,B 0,C 180,E1 -8963.98,E2 -8963.98} C_VEL
LIN {X 0,Y 441.28,Z 633.114,A -85,B 0,C 180,E1 -8965.32,E2 -8965.32} C_VEL
LIN {X 0,Y 440.455,Z 643.766,A -85,B 0,C 180,E1 -8966.872,E2 -8966.872} C_VEL
LIN {X 0,Y 439.819,Z 652.727,A -85,B 0,C 180,E1 -8968.444,E2 -8968.444} C_VEL
LIN {X 0,Y 439.239,Z 661.302,A -85,B 0,C 180,E1 -8970.263,E2 -8970.263} C_VEL
LIN {X 0,Y 438.829,Z 668.006,A -85,B 0,C 180,E1 -8972.027,E2 -8972.027} C_VEL
LIN {X 0,Y 438.585,Z 673.389,A -85,B 0,C 180,E1 -8973.815,E2 -8973.815} C_VEL
LIN {X 0,Y 438.375,Z 677.024,A -85,B 0,C 180,E1 -8975.365,E2 -8975.365} C_VEL
LIN {X 0,Y 438.285,Z 678.887,A -85,B 0,C 180,E1 -8976.366,E2 -8976.366} C_VEL
LIN {X 0,Y 438.193,Z 681.511,A -85,B 0,C 180,E1 -8978.353,E2 -8978.353} C_VEL
LIN {X 0,Y 438.151,Z 682.745,A -85,B 0,C 180,E1 -8980.315,E2 -8980.315} C_VEL
LIN {X 0,Y 438.189,Z 682.859,A -85,B 0,C 180,E1 -8981.29,E2 -8981.29} C_VEL
LIN {X 0,Y 438.158,Z 682.121,A -85,B 0,C 180,E1 -8983.219,E2 -8983.219} C_VEL
LIN {X 0,Y 438.255,Z 680.1,A -85,B 0,C 180,E1 -8985.132,E2 -8985.132} C_VEL
LIN {X 0,Y 438.43,Z 676.771,A -85,B 0,C 180,E1 -8987.031,E2 -8987.031} C_VEL
LIN {X 0,Y 438.668,Z 672.111,A -85,B 0,C 180,E1 -8988.915,E2 -8988.915} C_VEL
LIN {X 0,Y 438.967,Z 666.053,A -85,B 0,C 180,E1 -8990.787,E2 -8990.787} C_VEL
LIN {X 0,Y 439.53,Z 658.426,A -85,B 0,C 180,E1 -8992.65,E2 -8992.65} C_VEL
LIN {X 0,Y 440.112,Z 650.269,A -85,B 0,C 180,E1 -8994.272,E2 -8994.272} C_VEL
LIN {X 0,Y 440.885,Z 640.502,A -85,B 0,C 180,E1 -8995.886,E2 -8995.886} C_VEL
LIN {X 0,Y 441.714,Z 630.541,A -85,B 0,C 180,E1 -8997.264,E2 -8997.264} C_VEL
LIN {X 0,Y 442.637,Z 618.754,A -85,B 0,C 180,E1 -8998.635,E2 -8998.635} C_VEL
LIN {X 0,Y 443.631,Z 606.474,A -85,B 0,C 180,E1 -8999.821,E2 -8999.821} C_VEL
LIN {X 0,Y 444.645,Z 592.905,A -85,B 0,C 180,E1 -9000.905,E2 -9000.905} C_VEL
LIN {X 0,Y 445.573,Z 578.892,A -85,B 0,C 180,E1 -9001.807,E2 -9001.807} C_VEL
LIN {X 0,Y 446.384,Z 564.447,A -85,B 0,C 180,E1 -9002.538,E2 -9002.538} C_VEL
LIN {X 0,Y 447.034,Z 549.692,A -85,B 0,C 180,E1 -9003.098,E2 -9003.098} C_VEL
LIN {X 0,Y 447.517,Z 534.691,A -85,B 0,C 180,E1 -9003.489,E2 -9003.489} C_VEL
LIN {X 0,Y 450.204,Z 417.827,A -85,B 0,C 180,E1 -9005.696,E2 -9005.696} C_VEL
LIN {X 0,Y 450.586,Z 396.841,A -85,B 0,C 180,E1 -9006.122,E2 -9006.122} C_VEL
LIN {X 0,Y 448.06,Z 385.996,A -85,B 0,C 180,E1 -9006.532,E2 -9006.532} C_VEL
LIN {X 0,Y 443.16,Z 374.8,A -85,B 0,C 180,E1 -9007.16,E2 -9007.16} C_VEL
LIN {X 0,Y 440.405,Z 363.813,A -85,B 0,C 180,E1 -9009.646,E2 -9009.646} C_VEL
LIN {X 0,Y 439.456,Z 360.372,A -85,B 0,C 180,E1 -9010.481,E2 -9010.481} C_VEL
LIN {X 0,Y 439.471,Z 360.368,A -85,B 0,C 180,E1 -9012.937,E2 -9012.937} C_VEL
LIN {X 0,Y 439.451,Z 360.374,A -85,B 0,C 180,E1 -9016.347,E2 -9016.347} C_VEL
LIN {X 0,Y 439.407,Z 360.376,A -85,B 0,C 180,E1 -9019.626,E2 -9019.626} C_VEL
LIN {X 0,Y 439.368,Z 360.382,A -85,B 0,C 180,E1 -9022.575,E2 -9022.575} C_VEL
LIN {X 0,Y 439.369,Z 360.379,A -85,B 0,C 180,E1 -9025.587,E2 -9025.587} C_VEL
LIN {X 0,Y 439.385,Z 360.38,A -85,B 0,C 180,E1 -9028.676,E2 -9028.676} C_VEL
LIN {X 0,Y 439.367,Z 360.382,A -85,B 0,C 180,E1 -9032.028,E2 -9032.028} C_VEL
LIN {X 0,Y 439.389,Z 360.377,A -85,B 0,C 180,E1 -9035.338,E2 -9035.338} C_VEL
LIN {X 0,Y 439.353,Z 360.381,A -85,B 0,C 180,E1 -9038.598,E2 -9038.598} C_VEL
LIN {X 0,Y 439.361,Z 360.38,A -85,B 0,C 180,E1 -9041.251,E2 -9041.251} C_VEL
LIN {X 0,Y 439.374,Z 360.376,A -85,B 0,C 180,E1 -9044.733,E2 -9044.733} C_VEL
LIN {X 0,Y 439.347,Z 360.383,A -85,B 0,C 180,E1 -9047.789,E2 -9047.789} C_VEL
LIN {X 0,Y 439.35,Z 360.383,A -85,B 0,C 180,E1 -9051.4,E2 -9051.4} C_VEL
LIN {X 0,Y 439.388,Z 360.381,A -85,B 0,C 180,E1 -9054.842,E2 -9054.842} C_VEL
LIN {X 0,Y 439.365,Z 360.514,A -85,B 0,C 180,E1 -9057.491,E2 -9057.491} C_VEL
LIN {X 0,Y 442.655,Z 372.433,A -85,B 0,C 180,E1 -9059.991,E2 -9059.991} C_VEL
LIN {X 0,Y 445.336,Z 384.79,A -85,B 0,C 180,E1 -9062.362,E2 -9062.362} C_VEL
LIN {X 0,Y 444.586,Z 394.984,A -85,B 0,C 180,E1 -9063.989,E2 -9063.989} C_VEL
LIN {X 0,Y 448.192,Z 412.349,A -85,B 0,C 180,E1 -9064.631,E2 -9064.631} C_VEL
LIN {X 0,Y 450.342,Z 425.3,A -85,B 0,C 180,E1 -9065.053,E2 -9065.053} C_VEL
LIN {X 0,Y 447.645,Z 540.43,A -85,B 0,C 180,E1 -9067.225,E2 -9067.225} C_VEL
LIN {X 0,Y 447.065,Z 564.774,A -85,B 0,C 180,E1 -9067.711,E2 -9067.711} C_VEL
LIN {X 0,Y 446.309,Z 580.613,A -85,B 0,C 180,E1 -9068.21,E2 -9068.21} C_VEL
LIN {X 0,Y 445.468,Z 596.207,A -85,B 0,C 180,E1 -9068.904,E2 -9068.904} C_VEL
LIN {X 0,Y 444.637,Z 609.212,A -85,B 0,C 180,E1 -9069.65,E2 -9069.65} C_VEL
LIN {X 0,Y 443.669,Z 622.281,A -85,B 0,C 180,E1 -9070.569,E2 -9070.569} C_VEL
LIN {X 0,Y 442.62,Z 635.715,A -85,B 0,C 180,E1 -9071.723,E2 -9071.723} C_VEL
LIN {X 0,Y 441.657,Z 648.1,A -85,B 0,C 180,E1 -9073.01,E2 -9073.01} C_VEL
LIN {X 0,Y 440.822,Z 658.391,A -85,B 0,C 180,E1 -9074.273,E2 -9074.273} C_VEL
LIN {X 0,Y 440.168,Z 668.001,A -85,B 0,C 180,E1 -9075.67,E2 -9075.67} C_VEL
LIN {X 0,Y 439.382,Z 677.71,A -85,B 0,C 180,E1 -9077.344,E2 -9077.344} C_VEL
LIN {X 0,Y 439.074,Z 685.277,A -85,B 0,C 180,E1 -9078.925,E2 -9078.925} C_VEL
LIN {X 0,Y 438.635,Z 692.589,A -85,B 0,C 180,E1 -9080.779,E2 -9080.779} C_VEL
LIN {X 0,Y 438.431,Z 698.34,A -85,B 0,C 180,E1 -9082.631,E2 -9082.631} C_VEL
LIN {X 0,Y 438.316,Z 702.693,A -85,B 0,C 180,E1 -9084.478,E2 -9084.478} C_VEL
LIN {X 0,Y 438.236,Z 705.746,A -85,B 0,C 180,E1 -9086.321,E2 -9086.321} C_VEL
LIN {X 0,Y 438.292,Z 707.573,A -85,B 0,C 180,E1 -9088.161,E2 -9088.161} C_VEL
LIN {X 0,Y 438.25,Z 708.204,A -85,B 0,C 180,E1 -9089.999,E2 -9089.999} C_VEL
LIN {X 0,Y 438.292,Z 707.599,A -85,B 0,C 180,E1 -9091.836,E2 -9091.836} C_VEL
LIN {X 0,Y 438.259,Z 705.785,A -85,B 0,C 180,E1 -9093.676,E2 -9093.676} C_VEL
LIN {X 0,Y 438.324,Z 702.748,A -85,B 0,C 180,E1 -9095.519,E2 -9095.519} C_VEL
LIN {X 0,Y 438.485,Z 698.416,A -85,B 0,C 180,E1 -9097.365,E2 -9097.365} C_VEL
LIN {X 0,Y 438.644,Z 692.668,A -85,B 0,C 180,E1 -9099.218,E2 -9099.218} C_VEL
LIN {X 0,Y 439.086,Z 685.359,A -85,B 0,C 180,E1 -9101.072,E2 -9101.072} C_VEL
LIN {X 0,Y 439.461,Z 677.508,A -85,B 0,C 180,E1 -9102.702,E2 -9102.702} C_VEL
LIN {X 0,Y 440.154,Z 668.056,A -85,B 0,C 180,E1 -9104.327,E2 -9104.327} C_VEL
LIN {X 0,Y 440.848,Z 658.424,A -85,B 0,C 180,E1 -9105.723,E2 -9105.723} C_VEL
LIN {X 0,Y 441.772,Z 646.741,A -85,B 0,C 180,E1 -9107.139,E2 -9107.139} C_VEL
LIN {X 0,Y 442.665,Z 634.364,A -85,B 0,C 180,E1 -9108.392,E2 -9108.392} C_VEL
LIN {X 0,Y 443.773,Z 620.44,A -85,B 0,C 180,E1 -9109.544,E2 -9109.544} C_VEL
LIN {X 0,Y 444.694,Z 606.768,A -85,B 0,C 180,E1 -9110.465,E2 -9110.465} C_VEL
LIN {X 0,Y 445.622,Z 591.637,A -85,B 0,C 180,E1 -9111.267,E2 -9111.267} C_VEL
LIN {X 0,Y 446.32,Z 576.459,A -85,B 0,C 180,E1 -9111.872,E2 -9111.872} C_VEL
LIN {X 0,Y 446.918,Z 561.085,A -85,B 0,C 180,E1 -9112.293,E2 -9112.293} C_VEL
LIN {X 0,Y 449.447,Z 424.163,A -85,B 0,C 180,E1 -9114.745,E2 -9114.745} C_VEL
LIN {X 0,Y 444.118,Z 396.314,A -85,B 0,C 180,E1 -9115.597,E2 -9115.597} C_VEL
LIN {X 0,Y 444.968,Z 385.642,A -85,B 0,C 180,E1 -9117.259,E2 -9117.259} C_VEL
LIN {X 0,Y 444.475,Z 381.533,A -85,B 0,C 180,E1 -9117.952,E2 -9117.952} C_VEL
LIN {X 0,Y 440.98,Z 366.703,A -85,B 0,C 180,E1 -9120.615,E2 -9120.615} C_VEL
LIN {X 0,Y 439.38,Z 360.38,A -85,B 0,C 180,E1 -9121.79,E2 -9121.79} C_VEL
LIN {X 0,Y 439.385,Z 360.377,A -85,B 0,C 180,E1 -9125.155,E2 -9125.155} C_VEL
LIN {X 0,Y 439.345,Z 360.384,A -85,B 0,C 180,E1 -9128.597,E2 -9128.597} C_VEL
LIN {X 0,Y 439.347,Z 360.386,A -85,B 0,C 180,E1 -9132.208,E2 -9132.208} C_VEL
LIN {X 0,Y 439.364,Z 360.376,A -85,B 0,C 180,E1 -9135.266,E2 -9135.266} C_VEL
LIN {X 0,Y 439.351,Z 360.379,A -85,B 0,C 180,E1 -9138.746,E2 -9138.746} C_VEL
LIN {X 0,Y 439.343,Z 360.381,A -85,B 0,C 180,E1 -9141.61,E2 -9141.61} C_VEL
LIN {X 0,Y 439.381,Z 360.375,A -85,B 0,C 180,E1 -9144.843,E2 -9144.843} C_VEL
LIN {X 0,Y 439.359,Z 360.385,A -85,B 0,C 180,E1 -9148.139,E2 -9148.139} C_VEL
LIN {X 0,Y 439.368,Z 360.376,A -85,B 0,C 180,E1 -9151.323,E2 -9151.323} C_VEL
LIN {X 0,Y 439.351,Z 360.382,A -85,B 0,C 180,E1 -9154.412,E2 -9154.412} C_VEL
LIN {X 0,Y 439.347,Z 360.379,A -85,B 0,C 180,E1 -9157.424,E2 -9157.424} C_VEL
LIN {X 0,Y 439.426,Z 360.37,A -85,B 0,C 180,E1 -9160.663,E2 -9160.663} C_VEL
LIN {X 0,Y 439.403,Z 360.377,A -85,B 0,C 180,E1 -9164.223,E2 -9164.223} C_VEL
LIN {X 0,Y 439.469,Z 360.364,A -85,B 0,C 180,E1 -9167.285,E2 -9167.285} C_VEL
LIN {X 0,Y 439.474,Z 360.363,A -85,B 0,C 180,E1 -9170.798,E2 -9170.798} C_VEL
LIN {X 0,Y 439.545,Z 360.356,A -85,B 0,C 180,E1 -9173.574,E2 -9173.574} C_VEL
LIN {X 0,Y 439.391,Z 360.374,A -85,B 0,C 180,E1 -9175.413,E2 -9175.413} C_VEL
LIN {X 0,Y 439.61,Z 360.352,A -85,B 0,C 180,E1 -9178.168,E2 -9178.168} C_VEL
LIN {X 0,Y 439.672,Z 360.346,A -85,B 0,C 180,E1 -9180,E2 -9180} C_VEL
LIN {X 0,Y 439.587,Z 360.349,A -85,B 0,C 180,E1 -9182.749,E2 -9182.749} C_VEL
LIN {X 0,Y 439.543,Z 360.357,A -85,B 0,C 180,E1 -9186.427,E2 -9186.427} C_VEL
LIN {X 0,Y 439.466,Z 360.364,A -85,B 0,C 180,E1 -9189.203,E2 -9189.203} C_VEL
LIN {X 0,Y 439.45,Z 360.366,A -85,B 0,C 180,E1 -9192.938,E2 -9192.938} C_VEL
LIN {X 0,Y 439.388,Z 360.376,A -85,B 0,C 180,E1 -9196.329,E2 -9196.329} C_VEL
LIN {X 0,Y 439.388,Z 360.377,A -85,B 0,C 180,E1 -9199.627,E2 -9199.627} C_VEL
LIN {X 0,Y 439.348,Z 360.379,A -85,B 0,C 180,E1 -9202.577,E2 -9202.577} C_VEL
LIN {X 0,Y 439.353,Z 360.382,A -85,B 0,C 180,E1 -9205.588,E2 -9205.588} C_VEL
LIN {X 0,Y 439.369,Z 360.376,A -85,B 0,C 180,E1 -9208.677,E2 -9208.677} C_VEL
LIN {X 0,Y 439.357,Z 360.383,A -85,B 0,C 180,E1 -9212.031,E2 -9212.031} C_VEL
LIN {X 0,Y 439.381,Z 360.375,A -85,B 0,C 180,E1 -9215.158,E2 -9215.158} C_VEL
LIN {X 0,Y 439.344,Z 360.379,A -85,B 0,C 180,E1 -9218.599,E2 -9218.599} C_VEL
LIN {X 0,Y 439.339,Z 360.383,A -85,B 0,C 180,E1 -9222.212,E2 -9222.212} C_VEL
LIN {X 0,Y 439.367,Z 360.378,A -85,B 0,C 180,E1 -9225.269,E2 -9225.269} C_VEL
LIN {X 0,Y 439.356,Z 360.377,A -85,B 0,C 180,E1 -9228.749,E2 -9228.749} C_VEL
LIN {X 0,Y 439.35,Z 360.383,A -85,B 0,C 180,E1 -9231.612,E2 -9231.612} C_VEL
LIN {X 0,Y 439.388,Z 360.373,A -85,B 0,C 180,E1 -9234.845,E2 -9234.845} C_VEL
LIN {X 0,Y 439.367,Z 360.379,A -85,B 0,C 180,E1 -9238.141,E2 -9238.141} C_VEL
LIN {X 0,Y 439.396,Z 360.378,A -85,B 0,C 180,E1 -9241.608,E2 -9241.608} C_VEL
LIN {X 0,Y 439.362,Z 360.378,A -85,B 0,C 180,E1 -9244.414,E2 -9244.414} C_VEL
LIN {X 0,Y 439.362,Z 360.38,A -85,B 0,C 180,E1 -9247.426,E2 -9247.426} C_VEL
LIN {X 0,Y 439.44,Z 360.367,A -85,B 0,C 180,E1 -9250.665,E2 -9250.665} C_VEL
LIN {X 0,Y 439.461,Z 360.366,A -85,B 0,C 180,E1 -9254.226,E2 -9254.226} C_VEL
LIN {X 0,Y 439.484,Z 360.365,A -85,B 0,C 180,E1 -9258.003,E2 -9258.003} C_VEL
LIN {X 0,Y 439.503,Z 360.367,A -85,B 0,C 180,E1 -9261.727,E2 -9261.727} C_VEL
LIN {X 0,Y 439.6,Z 360.347,A -85,B 0,C 180,E1 -9264.497,E2 -9264.497} C_VEL
LIN {X 0,Y 439.629,Z 360.345,A -85,B 0,C 180,E1 -9268.169,E2 -9268.169} C_VEL
LIN {X 0,Y 439.691,Z 360.339,A -85,B 0,C 180,E1 -9270.001,E2 -9270.001} C_VEL
LIN {X 0,Y 439.504,Z 360.359,A -85,B 0,C 180,E1 -9270.957,E2 -9270.957} C_VEL
LIN {X 0,Y 438.86,Z 360.446,A -85,B 0,C 180,E1 -9271.722,E2 -9271.722} C_VEL
LIN {X 0,Y 435.923,Z 360.806,A -85,B 0,C 180,E1 -9272.962,E2 -9272.962} C_VEL
LIN {X 0,Y 433.463,Z 361.115,A -85,B 0,C 180,E1 -9273.964,E2 -9273.964} C_VEL
LIN {X 0,Y 432.478,Z 361.235,A -85,B 0,C 180,E1 -9274.739,E2 -9274.739} C_VEL
LIN {X 0,Y 432.439,Z 361.24,A -85,B 0,C 180,E1 -9275.001,E2 -9275.001} C_VEL
LIN {X 0,Y 432.518,Z 361.237,A -85,B 0,C 180,E1 -9277.608,E2 -9277.608} C_VEL
LIN {X 0,Y 432.408,Z 361.244,A -85,B 0,C 180,E1 -9280.3,E2 -9280.3} C_VEL
LIN {X 0,Y 432.404,Z 361.246,A -85,B 0,C 180,E1 -9283.154,E2 -9283.154} C_VEL
LIN {X 0,Y 432.366,Z 361.248,A -85,B 0,C 180,E1 -9286.456,E2 -9286.456} C_VEL
LIN {X 0,Y 432.392,Z 361.251,A -85,B 0,C 180,E1 -9289.486,E2 -9289.486} C_VEL
LIN {X 0,Y 432.318,Z 361.255,A -85,B 0,C 180,E1 -9292.965,E2 -9292.965} C_VEL
LIN {X 0,Y 432.323,Z 361.256,A -85,B 0,C 180,E1 -9296.036,E2 -9296.036} C_VEL
LIN {X 0,Y 432.333,Z 361.256,A -85,B 0,C 180,E1 -9299.189,E2 -9299.189} C_VEL
LIN {X 0,Y 432.329,Z 361.253,A -85,B 0,C 180,E1 -9302.444,E2 -9302.444} C_VEL
LIN {X 0,Y 432.349,Z 361.258,A -85,B 0,C 180,E1 -9305.632,E2 -9305.632} C_VEL
LIN {X 0,Y 432.332,Z 361.257,A -85,B 0,C 180,E1 -9308.712,E2 -9308.712} C_VEL
LIN {X 0,Y 432.357,Z 361.256,A -85,B 0,C 180,E1 -9312.423,E2 -9312.423} C_VEL
LIN {X 0,Y 432.353,Z 361.259,A -85,B 0,C 180,E1 -9312.582,E2 -9312.582} C_VEL
LIN {X 0,Y 435.13,Z 373.24,A -85,B 0,C 180,E1 -9314.976,E2 -9314.976} C_VEL
LIN {X 0,Y 440.765,Z 387.689,A -85,B 0,C 180,E1 -9315.598,E2 -9315.598} C_VEL
LIN {X 0,Y 443.131,Z 398.825,A -85,B 0,C 180,E1 -9315.952,E2 -9315.952} C_VEL
LIN {X 0,Y 440.297,Z 538.908,A -85,B 0,C 180,E1 -9318.52,E2 -9318.52} C_VEL
LIN {X 0,Y 439.71,Z 554.547,A -85,B 0,C 180,E1 -9318.992,E2 -9318.992} C_VEL
LIN {X 0,Y 438.933,Z 569.84,A -85,B 0,C 180,E1 -9319.649,E2 -9319.649} C_VEL
LIN {X 0,Y 438.091,Z 583.724,A -85,B 0,C 180,E1 -9320.428,E2 -9320.428} C_VEL
LIN {X 0,Y 437.155,Z 598.305,A -85,B 0,C 180,E1 -9321.465,E2 -9321.465} C_VEL
LIN {X 0,Y 436.194,Z 610.693,A -85,B 0,C 180,E1 -9322.538,E2 -9322.538} C_VEL
LIN {X 0,Y 435.223,Z 623.151,A -85,B 0,C 180,E1 -9323.844,E2 -9323.844} C_VEL
LIN {X 0,Y 434.296,Z 634.136,A -85,B 0,C 180,E1 -9325.219,E2 -9325.219} C_VEL
LIN {X 0,Y 433.411,Z 644.947,A -85,B 0,C 180,E1 -9326.847,E2 -9326.847} C_VEL
LIN {X 0,Y 432.772,Z 653.648,A -85,B 0,C 180,E1 -9328.417,E2 -9328.417} C_VEL
LIN {X 0,Y 432.158,Z 662.073,A -85,B 0,C 180,E1 -9330.263,E2 -9330.263} C_VEL
LIN {X 0,Y 431.792,Z 667.923,A -85,B 0,C 180,E1 -9331.835,E2 -9331.835} C_VEL
LIN {X 0,Y 431.519,Z 673.265,A -85,B 0,C 180,E1 -9333.609,E2 -9333.609} C_VEL
LIN {X 0,Y 431.341,Z 676.493,A -85,B 0,C 180,E1 -9334.936,E2 -9334.936} C_VEL
LIN {X 0,Y 431.137,Z 680.126,A -85,B 0,C 180,E1 -9336.969,E2 -9336.969} C_VEL
LIN {X 0,Y 431.084,Z 682.293,A -85,B 0,C 180,E1 -9338.981,E2 -9338.981} C_VEL
LIN {X 0,Y 431.093,Z 683.085,A -85,B 0,C 180,E1 -9341.009,E2 -9341.009} C_VEL
LIN {X 0,Y 431.062,Z 682.542,A -85,B 0,C 180,E1 -9342.934,E2 -9342.934} C_VEL
LIN {X 0,Y 431.14,Z 680.721,A -85,B 0,C 180,E1 -9344.881,E2 -9344.881} C_VEL
LIN {X 0,Y 431.306,Z 677.615,A -85,B 0,C 180,E1 -9346.813,E2 -9346.813} C_VEL
LIN {X 0,Y 431.55,Z 673.193,A -85,B 0,C 180,E1 -9348.73,E2 -9348.73} C_VEL
LIN {X 0,Y 431.872,Z 667.382,A -85,B 0,C 180,E1 -9350.634,E2 -9350.634} C_VEL
LIN {X 0,Y 432.427,Z 660.017,A -85,B 0,C 180,E1 -9352.529,E2 -9352.529} C_VEL
LIN {X 0,Y 433.052,Z 652.152,A -85,B 0,C 180,E1 -9354.178,E2 -9354.178} C_VEL
LIN {X 0,Y 433.826,Z 642.727,A -85,B 0,C 180,E1 -9355.819,E2 -9355.819} C_VEL
LIN {X 0,Y 434.707,Z 633.128,A -85,B 0,C 180,E1 -9357.22,E2 -9357.22} C_VEL
LIN {X 0,Y 435.603,Z 621.848,A -85,B 0,C 180,E1 -9358.613,E2 -9358.613} C_VEL
LIN {X 0,Y 436.657,Z 610.161,A -85,B 0,C 180,E1 -9359.818,E2 -9359.818} C_VEL
LIN {X 0,Y 437.719,Z 597.296,A -85,B 0,C 180,E1 -9360.92,E2 -9360.92} C_VEL
LIN {X 0,Y 438.654,Z 584.275,A -85,B 0,C 180,E1 -9361.836,E2 -9361.836} C_VEL
LIN {X 0,Y 439.611,Z 568.897,A -85,B 0,C 180,E1 -9362.691,E2 -9362.691} C_VEL
LIN {X 0,Y 440.359,Z 553.216,A -85,B 0,C 180,E1 -9363.345,E2 -9363.345} C_VEL
LIN {X 0,Y 440.958,Z 537.462,A -85,B 0,C 180,E1 -9363.798,E2 -9363.798} C_VEL
LIN {X 0,Y 444.184,Z 409.877,A -85,B 0,C 180,E1 -9366.285,E2 -9366.285} C_VEL
LIN {X 0,Y 444.387,Z 398.283,A -85,B 0,C 180,E1 -9366.525,E2 -9366.525} C_VEL
LIN {X 0,Y 442.28,Z 389.013,A -85,B 0,C 180,E1 -9366.892,E2 -9366.892} C_VEL
LIN {X 0,Y 436.087,Z 375.19,A -85,B 0,C 180,E1 -9367.699,E2 -9367.699} C_VEL
LIN {X 0,Y 433.197,Z 364.221,A -85,B 0,C 180,E1 -9370.28,E2 -9370.28} C_VEL
LIN {X 0,Y 432.397,Z 361.25,A -85,B 0,C 180,E1 -9371.069,E2 -9371.069} C_VEL
LIN {X 0,Y 432.405,Z 361.248,A -85,B 0,C 180,E1 -9373.152,E2 -9373.152} C_VEL
LIN {X 0,Y 432.417,Z 361.251,A -85,B 0,C 180,E1 -9376.478,E2 -9376.478} C_VEL
LIN {X 0,Y 432.343,Z 361.258,A -85,B 0,C 180,E1 -9379.96,E2 -9379.96} C_VEL
LIN {X 0,Y 432.316,Z 361.26,A -85,B 0,C 180,E1 -9382.964,E2 -9382.964} C_VEL
LIN {X 0,Y 432.321,Z 361.26,A -85,B 0,C 180,E1 -9386.035,E2 -9386.035} C_VEL
LIN {X 0,Y 432.326,Z 361.257,A -85,B 0,C 180,E1 -9389.188,E2 -9389.188} C_VEL
LIN {X 0,Y 432.324,Z 361.258,A -85,B 0,C 180,E1 -9392.443,E2 -9392.443} C_VEL
LIN {X 0,Y 432.336,Z 361.257,A -85,B 0,C 180,E1 -9395.818,E2 -9395.818} C_VEL
LIN {X 0,Y 432.302,Z 361.258,A -85,B 0,C 180,E1 -9399.348,E2 -9399.348} C_VEL
LIN {X 0,Y 432.303,Z 361.261,A -85,B 0,C 180,E1 -9401.8,E2 -9401.8} C_VEL
LIN {X 0,Y 432.334,Z 361.255,A -85,B 0,C 180,E1 -9404.347,E2 -9404.347} C_VEL
LIN {X 0,Y 432.304,Z 361.258,A -85,B 0,C 180,E1 -9407.018,E2 -9407.018} C_VEL
LIN {X 0,Y 432.29,Z 361.264,A -85,B 0,C 180,E1 -9409.827,E2 -9409.827} C_VEL
LIN {X 0,Y 432.296,Z 361.262,A -85,B 0,C 180,E1 -9413.02,E2 -9413.02} C_VEL
LIN {X 0,Y 432.332,Z 361.263,A -85,B 0,C 180,E1 -9416.002,E2 -9416.002} C_VEL
LIN {X 0,Y 432.32,Z 361.354,A -85,B 0,C 180,E1 -9416.933,E2 -9416.933} C_VEL
LIN {X 0,Y 435.598,Z 373.056,A -85,B 0,C 180,E1 -9419.491,E2 -9419.491} C_VEL
LIN {X 0,Y 438.54,Z 386.204,A -85,B 0,C 180,E1 -9422.098,E2 -9422.098} C_VEL
LIN {X 0,Y 438.21,Z 391.911,A -85,B 0,C 180,E1 -9423.058,E2 -9423.058} C_VEL
LIN {X 0,Y 437.974,Z 394.531,A -85,B 0,C 180,E1 -9423.481,E2 -9423.481} C_VEL
LIN {X 0,Y 441.769,Z 412.499,A -85,B 0,C 180,E1 -9424.177,E2 -9424.177} C_VEL
LIN {X 0,Y 444.029,Z 426.524,A -85,B 0,C 180,E1 -9424.65,E2 -9424.65} C_VEL
LIN {X 0,Y 441.149,Z 541.162,A -85,B 0,C 180,E1 -9426.87,E2 -9426.87} C_VEL
LIN {X 0,Y 440.532,Z 565.063,A -85,B 0,C 180,E1 -9427.363,E2 -9427.363} C_VEL
LIN {X 0,Y 439.713,Z 580.81,A -85,B 0,C 180,E1 -9427.872,E2 -9427.872} C_VEL
LIN {X 0,Y 438.824,Z 596.128,A -85,B 0,C 180,E1 -9428.569,E2 -9428.569} C_VEL
LIN {X 0,Y 437.844,Z 610.843,A -85,B 0,C 180,E1 -9429.443,E2 -9429.443} C_VEL
LIN {X 0,Y 436.729,Z 625,A -85,B 0,C 180,E1 -9430.492,E2 -9430.492} C_VEL
LIN {X 0,Y 435.615,Z 637.907,A -85,B 0,C 180,E1 -9431.662,E2 -9431.662} C_VEL
LIN {X 0,Y 434.665,Z 649.536,A -85,B 0,C 180,E1 -9432.928,E2 -9432.928} C_VEL
LIN {X 0,Y 433.791,Z 659.853,A -85,B 0,C 180,E1 -9434.253,E2 -9434.253} C_VEL
LIN {X 0,Y 432.968,Z 670.635,A -85,B 0,C 180,E1 -9435.907,E2 -9435.907} C_VEL
LIN {X 0,Y 432.327,Z 678.967,A -85,B 0,C 180,E1 -9437.429,E2 -9437.429} C_VEL
LIN {X 0,Y 431.901,Z 687.064,A -85,B 0,C 180,E1 -9439.213,E2 -9439.213} C_VEL
LIN {X 0,Y 431.492,Z 693.968,A -85,B 0,C 180,E1 -9441.097,E2 -9441.097} C_VEL
LIN {X 0,Y 431.315,Z 699.373,A -85,B 0,C 180,E1 -9442.979,E2 -9442.979} C_VEL
LIN {X 0,Y 431.229,Z 702.495,A -85,B 0,C 180,E1 -9444.387,E2 -9444.387} C_VEL
LIN {X 0,Y 431.144,Z 705.547,A -85,B 0,C 180,E1 -9446.26,E2 -9446.26} C_VEL
LIN {X 0,Y 431.214,Z 707.371,A -85,B 0,C 180,E1 -9448.131,E2 -9448.131} C_VEL
LIN {X 0,Y 431.164,Z 707.996,A -85,B 0,C 180,E1 -9449.999,E2 -9449.999} C_VEL
LIN {X 0,Y 431.215,Z 707.385,A -85,B 0,C 180,E1 -9451.867,E2 -9451.867} C_VEL
LIN {X 0,Y 431.165,Z 705.554,A -85,B 0,C 180,E1 -9453.737,E2 -9453.737} C_VEL
LIN {X 0,Y 431.235,Z 702.496,A -85,B 0,C 180,E1 -9455.61,E2 -9455.61} C_VEL
LIN {X 0,Y 431.384,Z 698.136,A -85,B 0,C 180,E1 -9457.487,E2 -9457.487} C_VEL
LIN {X 0,Y 431.586,Z 692.355,A -85,B 0,C 180,E1 -9459.37,E2 -9459.37} C_VEL
LIN {X 0,Y 432.066,Z 685.005,A -85,B 0,C 180,E1 -9461.254,E2 -9461.254} C_VEL
LIN {X 0,Y 432.398,Z 677.778,A -85,B 0,C 180,E1 -9462.785,E2 -9462.785} C_VEL
LIN {X 0,Y 433.069,Z 669.102,A -85,B 0,C 180,E1 -9464.327,E2 -9464.327} C_VEL
LIN {X 0,Y 433.939,Z 657.895,A -85,B 0,C 180,E1 -9465.98,E2 -9465.98} C_VEL
LIN {X 0,Y 434.918,Z 645.981,A -85,B 0,C 180,E1 -9467.436,E2 -9467.436} C_VEL
LIN {X 0,Y 435.846,Z 633.672,A -85,B 0,C 180,E1 -9468.69,E2 -9468.69} C_VEL
LIN {X 0,Y 436.879,Z 621.228,A -85,B 0,C 180,E1 -9469.743,E2 -9469.743} C_VEL
LIN {X 0,Y 437.834,Z 607.771,A -85,B 0,C 180,E1 -9470.678,E2 -9470.678} C_VEL
LIN {X 0,Y 438.78,Z 593.02,A -85,B 0,C 180,E1 -9471.492,E2 -9471.492} C_VEL
LIN {X 0,Y 439.569,Z 577.648,A -85,B 0,C 180,E1 -9472.132,E2 -9472.132} C_VEL
LIN {X 0,Y 440.212,Z 561.642,A -85,B 0,C 180,E1 -9472.59,E2 -9472.59} C_VEL
LIN {X 0,Y 442.957,Z 425.614,A -85,B 0,C 180,E1 -9475.073,E2 -9475.073} C_VEL
LIN {X 0,Y 437.371,Z 396.152,A -85,B 0,C 180,E1 -9475.992,E2 -9475.992} C_VEL
LIN {X 0,Y 438.136,Z 386.852,A -85,B 0,C 180,E1 -9477.461,E2 -9477.461} C_VEL
LIN {X 0,Y 437.324,Z 381.862,A -85,B 0,C 180,E1 -9478.329,E2 -9478.329} C_VEL
LIN {X 0,Y 434.004,Z 367.939,A -85,B 0,C 180,E1 -9480.88,E2 -9480.88} C_VEL
LIN {X 0,Y 432.326,Z 361.258,A -85,B 0,C 180,E1 -9482.165,E2 -9482.165} C_VEL
LIN {X 0,Y 432.327,Z 361.257,A -85,B 0,C 180,E1 -9484.676,E2 -9484.676} C_VEL
LIN {X 0,Y 432.313,Z 361.262,A -85,B 0,C 180,E1 -9488.15,E2 -9488.15} C_VEL
LIN {X 0,Y 432.298,Z 361.26,A -85,B 0,C 180,E1 -9491.799,E2 -9491.799} C_VEL
LIN {X 0,Y 432.321,Z 361.259,A -85,B 0,C 180,E1 -9494.346,E2 -9494.346} C_VEL
LIN {X 0,Y 432.291,Z 361.258,A -85,B 0,C 180,E1 -9497.017,E2 -9497.017} C_VEL
LIN {X 0,Y 432.276,Z 361.263,A -85,B 0,C 180,E1 -9499.827,E2 -9499.827} C_VEL
LIN {X 0,Y 432.283,Z 361.259,A -85,B 0,C 180,E1 -9503.02,E2 -9503.02} C_VEL
LIN {X 0,Y 432.345,Z 361.257,A -85,B 0,C 180,E1 -9505.996,E2 -9505.996} C_VEL
LIN {X 0,Y 432.332,Z 361.253,A -85,B 0,C 180,E1 -9509.489,E2 -9509.489} C_VEL
LIN {X 0,Y 432.305,Z 361.26,A -85,B 0,C 180,E1 -9511.872,E2 -9511.872} C_VEL
LIN {X 0,Y 432.309,Z 361.255,A -85,B 0,C 180,E1 -9514.996,E2 -9514.996} C_VEL
LIN {X 0,Y 432.342,Z 361.258,A -85,B 0,C 180,E1 -9518.045,E2 -9518.045} C_VEL
LIN {X 0,Y 432.366,Z 361.248,A -85,B 0,C 180,E1 -9521.029,E2 -9521.029} C_VEL
LIN {X 0,Y 432.373,Z 361.254,A -85,B 0,C 180,E1 -9523.959,E2 -9523.959} C_VEL
LIN {X 0,Y 432.443,Z 361.243,A -85,B 0,C 180,E1 -9527.803,E2 -9527.803} C_VEL
LIN {X 0,Y 432.446,Z 361.241,A -85,B 0,C 180,E1 -9531.59,E2 -9531.59} C_VEL
LIN {X 0,Y 432.557,Z 361.227,A -85,B 0,C 180,E1 -9534.406,E2 -9534.406} C_VEL
LIN {X 0,Y 432.579,Z 361.228,A -85,B 0,C 180,E1 -9538.138,E2 -9538.138} C_VEL
LIN {X 0,Y 432.623,Z 361.224,A -85,B 0,C 180,E1 -9540,E2 -9540} C_VEL
LIN {X 0,Y 432.541,Z 361.227,A -85,B 0,C 180,E1 -9542.794,E2 -9542.794} C_VEL
LIN {X 0,Y 432.555,Z 361.228,A -85,B 0,C 180,E1 -9545.595,E2 -9545.595} C_VEL
LIN {X 0,Y 432.434,Z 361.242,A -85,B 0,C 180,E1 -9548.411,E2 -9548.411} C_VEL
LIN {X 0,Y 432.439,Z 361.244,A -85,B 0,C 180,E1 -9552.197,E2 -9552.197} C_VEL
LIN {X 0,Y 432.374,Z 361.254,A -85,B 0,C 180,E1 -9556.041,E2 -9556.041} C_VEL
LIN {X 0,Y 432.373,Z 361.25,A -85,B 0,C 180,E1 -9559.486,E2 -9559.486} C_VEL
LIN {X 0,Y 432.297,Z 361.257,A -85,B 0,C 180,E1 -9562.966,E2 -9562.966} C_VEL
LIN {X 0,Y 432.305,Z 361.262,A -85,B 0,C 180,E1 -9566.037,E2 -9566.037} C_VEL
LIN {X 0,Y 432.311,Z 361.256,A -85,B 0,C 180,E1 -9569.19,E2 -9569.19} C_VEL
LIN {X 0,Y 432.311,Z 361.256,A -85,B 0,C 180,E1 -9572.444,E2 -9572.444} C_VEL
LIN {X 0,Y 432.329,Z 361.258,A -85,B 0,C 180,E1 -9575.632,E2 -9575.632} C_VEL
LIN {X 0,Y 432.308,Z 361.255,A -85,B 0,C 180,E1 -9578.712,E2 -9578.712} C_VEL
LIN {X 0,Y 432.293,Z 361.265,A -85,B 0,C 180,E1 -9581.802,E2 -9581.802} C_VEL
LIN {X 0,Y 432.323,Z 361.255,A -85,B 0,C 180,E1 -9584.349,E2 -9584.349} C_VEL
LIN {X 0,Y 432.295,Z 361.257,A -85,B 0,C 180,E1 -9587.02,E2 -9587.02} C_VEL
LIN {X 0,Y 432.281,Z 361.267,A -85,B 0,C 180,E1 -9589.83,E2 -9589.83} C_VEL
LIN {X 0,Y 432.292,Z 361.258,A -85,B 0,C 180,E1 -9593.023,E2 -9593.023} C_VEL
LIN {X 0,Y 432.338,Z 361.257,A -85,B 0,C 180,E1 -9596.001,E2 -9596.001} C_VEL
LIN {X 0,Y 432.342,Z 361.255,A -85,B 0,C 180,E1 -9599.492,E2 -9599.492} C_VEL
LIN {X 0,Y 432.323,Z 361.26,A -85,B 0,C 180,E1 -9601.875,E2 -9601.875} C_VEL
LIN {X 0,Y 432.347,Z 361.256,A -85,B 0,C 180,E1 -9605.549,E2 -9605.549} C_VEL
LIN {X 0,Y 432.348,Z 361.251,A -85,B 0,C 180,E1 -9609.048,E2 -9609.048} C_VEL
LIN {X 0,Y 432.357,Z 361.253,A -85,B 0,C 180,E1 -9612.012,E2 -9612.012} C_VEL
LIN {X 0,Y 432.393,Z 361.245,A -85,B 0,C 180,E1 -9614.928,E2 -9614.928} C_VEL
LIN {X 0,Y 432.46,Z 361.243,A -85,B 0,C 180,E1 -9617.805,E2 -9617.805} C_VEL
LIN {X 0,Y 432.463,Z 361.243,A -85,B 0,C 180,E1 -9621.591,E2 -9621.591} C_VEL
LIN {X 0,Y 432.555,Z 361.225,A -85,B 0,C 180,E1 -9624.407,E2 -9624.407} C_VEL
LIN {X 0,Y 432.598,Z 361.221,A -85,B 0,C 180,E1 -9628.139,E2 -9628.139} C_VEL
LIN {X 0,Y 432.642,Z 361.217,A -85,B 0,C 180,E1 -9630.001,E2 -9630.001} C_VEL
LIN {X 0,Y 432.564,Z 361.224,A -85,B 0,C 180,E1 -9632.795,E2 -9632.795} C_VEL
LIN {X 0,Y 432.439,Z 361.24,A -85,B 0,C 180,E1 -9635.001,E2 -9635.001} C_VEL
LIN {X 0,Y 431.874,Z 361.315,A -85,B 0,C 180,E1 -9635.78,E2 -9635.78} C_VEL
LIN {X 0,Y 429.023,Z 361.666,A -85,B 0,C 180,E1 -9637.044,E2 -9637.044} C_VEL
LIN {X 0,Y 426.544,Z 361.976,A -85,B 0,C 180,E1 -9638.065,E2 -9638.065} C_VEL
LIN {X 0,Y 425.476,Z 362.107,A -85,B 0,C 180,E1 -9638.854,E2 -9638.854} C_VEL
LIN {X 0,Y 425.392,Z 362.119,A -85,B 0,C 180,E1 -9639.122,E2 -9639.122} C_VEL
LIN {X 0,Y 425.399,Z 362.117,A -85,B 0,C 180,E1 -9642.905,E2 -9642.905} C_VEL
LIN {X 0,Y 425.323,Z 362.125,A -85,B 0,C 180,E1 -9646.586,E2 -9646.586} C_VEL
LIN {X 0,Y 425.334,Z 362.131,A -85,B 0,C 180,E1 -9649.636,E2 -9649.636} C_VEL
LIN {X 0,Y 425.293,Z 362.13,A -85,B 0,C 180,E1 -9652.34,E2 -9652.34} C_VEL
LIN {X 0,Y 425.266,Z 362.139,A -85,B 0,C 180,E1 -9655.448,E2 -9655.448} C_VEL
LIN {X 0,Y 425.313,Z 362.128,A -85,B 0,C 180,E1 -9658.861,E2 -9658.861} C_VEL
LIN {X 0,Y 425.271,Z 362.135,A -85,B 0,C 180,E1 -9661.928,E2 -9661.928} C_VEL
LIN {X 0,Y 425.305,Z 362.133,A -85,B 0,C 180,E1 -9665.337,E2 -9665.337} C_VEL
LIN {X 0,Y 425.287,Z 362.135,A -85,B 0,C 180,E1 -9668.901,E2 -9668.901} C_VEL
LIN {X 0,Y 425.332,Z 362.17,A -85,B 0,C 180,E1 -9672.26,E2 -9672.26} C_VEL
LIN {X 0,Y 427.84,Z 373.096,A -85,B 0,C 180,E1 -9674.526,E2 -9674.526} C_VEL
LIN {X 0,Y 434.562,Z 390.257,A -85,B 0,C 180,E1 -9675.29,E2 -9675.29} C_VEL
LIN {X 0,Y 436.588,Z 399.486,A -85,B 0,C 180,E1 -9675.594,E2 -9675.594} C_VEL
LIN {X 0,Y 433.623,Z 539.102,A -85,B 0,C 180,E1 -9678.208,E2 -9678.208} C_VEL
LIN {X 0,Y 433.008,Z 554.802,A -85,B 0,C 180,E1 -9678.69,E2 -9678.69} C_VEL
LIN {X 0,Y 432.209,Z 569.934,A -85,B 0,C 180,E1 -9679.349,E2 -9679.349} C_VEL
LIN {X 0,Y 431.375,Z 583.522,A -85,B 0,C 180,E1 -9680.12,E2 -9680.12} C_VEL
LIN {X 0,Y 430.341,Z 598.423,A -85,B 0,C 180,E1 -9681.192,E2 -9681.192} C_VEL
LIN {X 0,Y 429.367,Z 610.831,A -85,B 0,C 180,E1 -9682.282,E2 -9682.282} C_VEL
LIN {X 0,Y 428.376,Z 623.085,A -85,B 0,C 180,E1 -9683.582,E2 -9683.582} C_VEL
LIN {X 0,Y 427.354,Z 634.364,A -85,B 0,C 180,E1 -9685.012,E2 -9685.012} C_VEL
LIN {X 0,Y 426.53,Z 644.175,A -85,B 0,C 180,E1 -9686.496,E2 -9686.496} C_VEL
LIN {X 0,Y 425.814,Z 653.156,A -85,B 0,C 180,E1 -9688.119,E2 -9688.119} C_VEL
LIN {X 0,Y 425.165,Z 661.778,A -85,B 0,C 180,E1 -9690.003,E2 -9690.003} C_VEL
LIN {X 0,Y 424.717,Z 668.61,A -85,B 0,C 180,E1 -9691.861,E2 -9691.861} C_VEL
LIN {X 0,Y 424.472,Z 673.267,A -85,B 0,C 180,E1 -9693.446,E2 -9693.446} C_VEL
LIN {X 0,Y 424.182,Z 677.988,A -85,B 0,C 180,E1 -9695.53,E2 -9695.53} C_VEL
LIN {X 0,Y 424.013,Z 681.146,A -85,B 0,C 180,E1 -9697.59,E2 -9697.59} C_VEL
LIN {X 0,Y 423.964,Z 682.869,A -85,B 0,C 180,E1 -9699.628,E2 -9699.628} C_VEL
LIN {X 0,Y 423.976,Z 683.233,A -85,B 0,C 180,E1 -9701.642,E2 -9701.642} C_VEL
LIN {X 0,Y 424.01,Z 682.29,A -85,B 0,C 180,E1 -9703.633,E2 -9703.633} C_VEL
LIN {X 0,Y 424.076,Z 680.069,A -85,B 0,C 180,E1 -9705.606,E2 -9705.606} C_VEL
LIN {X 0,Y 424.349,Z 676.538,A -85,B 0,C 180,E1 -9707.566,E2 -9707.566} C_VEL
LIN {X 0,Y 424.583,Z 671.684,A -85,B 0,C 180,E1 -9709.509,E2 -9709.509} C_VEL
LIN {X 0,Y 425.038,Z 665.381,A -85,B 0,C 180,E1 -9711.441,E2 -9711.441} C_VEL
LIN {X 0,Y 425.521,Z 659.01,A -85,B 0,C 180,E1 -9713.025,E2 -9713.025} C_VEL
LIN {X 0,Y 426.288,Z 650.366,A -85,B 0,C 180,E1 -9714.797,E2 -9714.797} C_VEL
LIN {X 0,Y 427.147,Z 640.556,A -85,B 0,C 180,E1 -9716.462,E2 -9716.462} C_VEL
LIN {X 0,Y 428.087,Z 630.519,A -85,B 0,C 180,E1 -9717.883,E2 -9717.883} C_VEL
LIN {X 0,Y 429.16,Z 619.228,A -85,B 0,C 180,E1 -9719.227,E2 -9719.227} C_VEL
LIN {X 0,Y 430.255,Z 606.772,A -85,B 0,C 180,E1 -9720.468,E2 -9720.468} C_VEL
LIN {X 0,Y 431.304,Z 594.019,A -85,B 0,C 180,E1 -9721.517,E2 -9721.517} C_VEL
LIN {X 0,Y 432.332,Z 580.208,A -85,B 0,C 180,E1 -9722.445,E2 -9722.445} C_VEL
LIN {X 0,Y 433.234,Z 566.089,A -85,B 0,C 180,E1 -9723.196,E2 -9723.196} C_VEL
LIN {X 0,Y 433.986,Z 551.062,A -85,B 0,C 180,E1 -9723.801,E2 -9723.801} C_VEL
LIN {X 0,Y 434.565,Z 535.468,A -85,B 0,C 180,E1 -9724.231,E2 -9724.231} C_VEL
LIN {X 0,Y 437.622,Z 422.105,A -85,B 0,C 180,E1 -9726.483,E2 -9726.483} C_VEL
LIN {X 0,Y 438.152,Z 399.39,A -85,B 0,C 180,E1 -9726.968,E2 -9726.968} C_VEL
LIN {X 0,Y 436.307,Z 391.524,A -85,B 0,C 180,E1 -9727.291,E2 -9727.291} C_VEL
LIN {X 0,Y 430.11,Z 378.084,A -85,B 0,C 180,E1 -9728.125,E2 -9728.125} C_VEL
LIN {X 0,Y 428.965,Z 375.497,A -85,B 0,C 180,E1 -9728.301,E2 -9728.301} C_VEL
LIN {X 0,Y 426.599,Z 366.695,A -85,B 0,C 180,E1 -9730.441,E2 -9730.441} C_VEL
LIN {X 0,Y 425.367,Z 362.124,A -85,B 0,C 180,E1 -9731.617,E2 -9731.617} C_VEL
LIN {X 0,Y 425.352,Z 362.13,A -85,B 0,C 180,E1 -9734.35,E2 -9734.35} C_VEL
LIN {X 0,Y 425.338,Z 362.13,A -85,B 0,C 180,E1 -9737.302,E2 -9737.302} C_VEL
LIN {X 0,Y 425.3,Z 362.135,A -85,B 0,C 180,E1 -9740.305,E2 -9740.305} C_VEL
LIN {X 0,Y 425.277,Z 362.136,A -85,B 0,C 180,E1 -9743.367,E2 -9743.367} C_VEL
LIN {X 0,Y 425.29,Z 362.135,A -85,B 0,C 180,E1 -9746.499,E2 -9746.499} C_VEL
LIN {X 0,Y 425.283,Z 362.135,A -85,B 0,C 180,E1 -9749.72,E2 -9749.72} C_VEL
LIN {X 0,Y 425.272,Z 362.135,A -85,B 0,C 180,E1 -9753.049,E2 -9753.049} C_VEL
LIN {X 0,Y 425.279,Z 362.136,A -85,B 0,C 180,E1 -9755.927,E2 -9755.927} C_VEL
LIN {X 0,Y 425.259,Z 362.136,A -85,B 0,C 180,E1 -9759.035,E2 -9759.035} C_VEL
LIN {X 0,Y 425.257,Z 362.137,A -85,B 0,C 180,E1 -9762.655,E2 -9762.655} C_VEL
LIN {X 0,Y 425.286,Z 362.131,A -85,B 0,C 180,E1 -9765.283,E2 -9765.283} C_VEL
LIN {X 0,Y 425.248,Z 362.137,A -85,B 0,C 180,E1 -9768.617,E2 -9768.617} C_VEL
LIN {X 0,Y 425.27,Z 362.138,A -85,B 0,C 180,E1 -9772.304,E2 -9772.304} C_VEL
LIN {X 0,Y 425.284,Z 362.14,A -85,B 0,C 180,E1 -9775.814,E2 -9775.814} C_VEL
LIN {X 0,Y 425.288,Z 362.242,A -85,B 0,C 180,E1 -9776.349,E2 -9776.349} C_VEL
LIN {X 0,Y 428.688,Z 374.195,A -85,B 0,C 180,E1 -9779.063,E2 -9779.063} C_VEL
LIN {X 0,Y 431.501,Z 386.468,A -85,B 0,C 180,E1 -9781.584,E2 -9781.584} C_VEL
LIN {X 0,Y 431.936,Z 389.198,A -85,B 0,C 180,E1 -9782.108,E2 -9782.108} C_VEL
LIN {X 0,Y 431.441,Z 394.072,A -85,B 0,C 180,E1 -9782.932,E2 -9782.932} C_VEL
LIN {X 0,Y 435.491,Z 413.124,A -85,B 0,C 180,E1 -9783.722,E2 -9783.722} C_VEL
LIN {X 0,Y 437.777,Z 427.351,A -85,B 0,C 180,E1 -9784.219,E2 -9784.219} C_VEL
LIN {X 0,Y 434.836,Z 536.102,A -85,B 0,C 180,E1 -9786.388,E2 -9786.388} C_VEL
LIN {X 0,Y 434.112,Z 563.421,A -85,B 0,C 180,E1 -9786.946,E2 -9786.946} C_VEL
LIN {X 0,Y 433.247,Z 578.921,A -85,B 0,C 180,E1 -9787.436,E2 -9787.436} C_VEL
LIN {X 0,Y 432.35,Z 593.919,A -85,B 0,C 180,E1 -9788.107,E2 -9788.107} C_VEL
LIN {X 0,Y 431.264,Z 609.022,A -85,B 0,C 180,E1 -9788.99,E2 -9788.99} C_VEL
LIN {X 0,Y 430.089,Z 623.449,A -85,B 0,C 180,E1 -9790.054,E2 -9790.054} C_VEL
LIN {X 0,Y 428.94,Z 636.568,A -85,B 0,C 180,E1 -9791.242,E2 -9791.242} C_VEL
LIN {X 0,Y 427.832,Z 648.978,A -85,B 0,C 180,E1 -9792.598,E2 -9792.598} C_VEL
LIN {X 0,Y 426.874,Z 659.677,A -85,B 0,C 180,E1 -9793.991,E2 -9793.991} C_VEL
LIN {X 0,Y 426.004,Z 670.448,A -85,B 0,C 180,E1 -9795.671,E2 -9795.671} C_VEL
LIN {X 0,Y 425.295,Z 679.304,A -85,B 0,C 180,E1 -9797.328,E2 -9797.328} C_VEL
LIN {X 0,Y 424.883,Z 686.874,A -85,B 0,C 180,E1 -9799.033,E2 -9799.033} C_VEL
LIN {X 0,Y 424.439,Z 693.776,A -85,B 0,C 180,E1 -9800.948,E2 -9800.948} C_VEL
LIN {X 0,Y 424.236,Z 699.183,A -85,B 0,C 180,E1 -9802.861,E2 -9802.861} C_VEL
LIN {X 0,Y 424.148,Z 702.304,A -85,B 0,C 180,E1 -9804.293,E2 -9804.293} C_VEL
LIN {X 0,Y 424.056,Z 705.354,A -85,B 0,C 180,E1 -9806.198,E2 -9806.198} C_VEL
LIN {X 0,Y 424.139,Z 707.171,A -85,B 0,C 180,E1 -9808.099,E2 -9808.099} C_VEL
LIN {X 0,Y 424.081,Z 707.785,A -85,B 0,C 180,E1 -9809.999,E2 -9809.999} C_VEL
LIN {X 0,Y 424.139,Z 707.167,A -85,B 0,C 180,E1 -9811.898,E2 -9811.898} C_VEL
LIN {X 0,Y 424.076,Z 705.316,A -85,B 0,C 180,E1 -9813.799,E2 -9813.799} C_VEL
LIN {X 0,Y 424.15,Z 702.234,A -85,B 0,C 180,E1 -9815.704,E2 -9815.704} C_VEL
LIN {X 0,Y 424.306,Z 697.844,A -85,B 0,C 180,E1 -9817.613,E2 -9817.613} C_VEL
LIN {X 0,Y 424.518,Z 692.027,A -85,B 0,C 180,E1 -9819.528,E2 -9819.528} C_VEL
LIN {X 0,Y 425.01,Z 684.635,A -85,B 0,C 180,E1 -9821.444,E2 -9821.444} C_VEL
LIN {X 0,Y 425.412,Z 677.186,A -85,B 0,C 180,E1 -9823.032,E2 -9823.032} C_VEL
LIN {X 0,Y 426.104,Z 668.632,A -85,B 0,C 180,E1 -9824.566,E2 -9824.566} C_VEL
LIN {X 0,Y 426.854,Z 659.101,A -85,B 0,C 180,E1 -9826.007,E2 -9826.007} C_VEL
LIN {X 0,Y 427.812,Z 648.095,A -85,B 0,C 180,E1 -9827.41,E2 -9827.41} C_VEL
LIN {X 0,Y 428.814,Z 635.451,A -85,B 0,C 180,E1 -9828.761,E2 -9828.761} C_VEL
LIN {X 0,Y 429.991,Z 621.881,A -85,B 0,C 180,E1 -9829.948,E2 -9829.948} C_VEL
LIN {X 0,Y 430.975,Z 608.579,A -85,B 0,C 180,E1 -9830.897,E2 -9830.897} C_VEL
LIN {X 0,Y 431.976,Z 594.112,A -85,B 0,C 180,E1 -9831.722,E2 -9831.722} C_VEL
LIN {X 0,Y 432.756,Z 578.967,A -85,B 0,C 180,E1 -9832.383,E2 -9832.383} C_VEL
LIN {X 0,Y 433.473,Z 563.216,A -85,B 0,C 180,E1 -9832.863,E2 -9832.863} C_VEL
LIN {X 0,Y 436.365,Z 426.353,A -85,B 0,C 180,E1 -9835.423,E2 -9835.423} C_VEL
LIN {X 0,Y 430.639,Z 395.986,A -85,B 0,C 180,E1 -9836.392,E2 -9836.392} C_VEL
LIN {X 0,Y 431.22,Z 387.007,A -85,B 0,C 180,E1 -9837.847,E2 -9837.847} C_VEL
LIN {X 0,Y 428.47,Z 374.894,A -85,B 0,C 180,E1 -9840.065,E2 -9840.065} C_VEL
LIN {X 0,Y 425.283,Z 362.137,A -85,B 0,C 180,E1 -9842.514,E2 -9842.514} C_VEL
LIN {X 0,Y 425.287,Z 362.134,A -85,B 0,C 180,E1 -9845.335,E2 -9845.335} C_VEL
LIN {X 0,Y 425.266,Z 362.136,A -85,B 0,C 180,E1 -9848.9,E2 -9848.9} C_VEL
LIN {X 0,Y 425.249,Z 362.137,A -85,B 0,C 180,E1 -9852.654,E2 -9852.654} C_VEL
LIN {X 0,Y 425.272,Z 362.132,A -85,B 0,C 180,E1 -9855.282,E2 -9855.282} C_VEL
LIN {X 0,Y 425.236,Z 362.139,A -85,B 0,C 180,E1 -9858.617,E2 -9858.617} C_VEL
LIN {X 0,Y 425.263,Z 362.133,A -85,B 0,C 180,E1 -9861.098,E2 -9861.098} C_VEL
LIN {X 0,Y 425.283,Z 362.132,A -85,B 0,C 180,E1 -9864.663,E2 -9864.663} C_VEL
LIN {X 0,Y 425.252,Z 362.141,A -85,B 0,C 180,E1 -9868.072,E2 -9868.072} C_VEL
LIN {X 0,Y 425.282,Z 362.131,A -85,B 0,C 180,E1 -9871.364,E2 -9871.364} C_VEL
LIN {X 0,Y 425.245,Z 362.138,A -85,B 0,C 180,E1 -9874.552,E2 -9874.552} C_VEL
LIN {X 0,Y 425.277,Z 362.134,A -85,B 0,C 180,E1 -9877.729,E2 -9877.729} C_VEL
LIN {X 0,Y 425.345,Z 362.124,A -85,B 0,C 180,E1 -9880.703,E2 -9880.703} C_VEL
LIN {X 0,Y 425.307,Z 362.13,A -85,B 0,C 180,E1 -9883.685,E2 -9883.685} C_VEL
LIN {X 0,Y 425.378,Z 362.119,A -85,B 0,C 180,E1 -9887.096,E2 -9887.096} C_VEL
LIN {X 0,Y 425.378,Z 362.121,A -85,B 0,C 180,E1 -9890.49,E2 -9890.49} C_VEL
LIN {X 0,Y 425.462,Z 362.109,A -85,B 0,C 180,E1 -9893.36,E2 -9893.36} C_VEL
LIN {X 0,Y 425.331,Z 362.125,A -85,B 0,C 180,E1 -9895.261,E2 -9895.261} C_VEL
LIN {X 0,Y 425.548,Z 362.104,A -85,B 0,C 180,E1 -9898.107,E2 -9898.107} C_VEL
LIN {X 0,Y 425.574,Z 362.102,A -85,B 0,C 180,E1 -9900,E2 -9900} C_VEL
LIN {X 0,Y 425.496,Z 362.104,A -85,B 0,C 180,E1 -9902.841,E2 -9902.841} C_VEL
LIN {X 0,Y 425.46,Z 362.109,A -85,B 0,C 180,E1 -9906.514,E2 -9906.514} C_VEL
LIN {X 0,Y 425.37,Z 362.122,A -85,B 0,C 180,E1 -9909.51,E2 -9909.51} C_VEL
LIN {X 0,Y 425.378,Z 362.119,A -85,B 0,C 180,E1 -9912.904,E2 -9912.904} C_VEL
LIN {X 0,Y 425.303,Z 362.129,A -85,B 0,C 180,E1 -9916.585,E2 -9916.585} C_VEL
LIN {X 0,Y 425.315,Z 362.13,A -85,B 0,C 180,E1 -9919.636,E2 -9919.636} C_VEL
LIN {X 0,Y 425.274,Z 362.134,A -85,B 0,C 180,E1 -9922.34,E2 -9922.34} C_VEL
LIN {X 0,Y 425.246,Z 362.137,A -85,B 0,C 180,E1 -9925.449,E2 -9925.449} C_VEL
LIN {X 0,Y 425.288,Z 362.13,A -85,B 0,C 180,E1 -9928.86,E2 -9928.86} C_VEL
LIN {X 0,Y 425.253,Z 362.141,A -85,B 0,C 180,E1 -9931.928,E2 -9931.928} C_VEL
LIN {X 0,Y 425.284,Z 362.132,A -85,B 0,C 180,E1 -9935.338,E2 -9935.338} C_VEL
LIN {X 0,Y 425.266,Z 362.133,A -85,B 0,C 180,E1 -9938.903,E2 -9938.903} C_VEL
LIN {X 0,Y 425.247,Z 362.135,A -85,B 0,C 180,E1 -9942.657,E2 -9942.657} C_VEL
LIN {X 0,Y 425.275,Z 362.133,A -85,B 0,C 180,E1 -9945.285,E2 -9945.285} C_VEL
LIN {X 0,Y 425.241,Z 362.136,A -85,B 0,C 180,E1 -9948.62,E2 -9948.62} C_VEL
LIN {X 0,Y 425.269,Z 362.133,A -85,B 0,C 180,E1 -9951.101,E2 -9951.101} C_VEL
LIN {X 0,Y 425.29,Z 362.13,A -85,B 0,C 180,E1 -9954.665,E2 -9954.665} C_VEL
LIN {X 0,Y 425.259,Z 362.137,A -85,B 0,C 180,E1 -9958.075,E2 -9958.075} C_VEL
LIN {X 0,Y 425.3,Z 362.131,A -85,B 0,C 180,E1 -9961.368,E2 -9961.368} C_VEL
LIN {X 0,Y 425.255,Z 362.134,A -85,B 0,C 180,E1 -9964.554,E2 -9964.554} C_VEL
LIN {X 0,Y 425.29,Z 362.137,A -85,B 0,C 180,E1 -9967.731,E2 -9967.731} C_VEL
LIN {X 0,Y 425.36,Z 362.121,A -85,B 0,C 180,E1 -9970.706,E2 -9970.706} C_VEL
LIN {X 0,Y 425.387,Z 362.125,A -85,B 0,C 180,E1 -9973.69,E2 -9973.69} C_VEL
LIN {X 0,Y 425.413,Z 362.121,A -85,B 0,C 180,E1 -9977.6,E2 -9977.6} C_VEL
LIN {X 0,Y 425.408,Z 362.12,A -85,B 0,C 180,E1 -9981.451,E2 -9981.451} C_VEL
LIN {X 0,Y 425.512,Z 362.103,A -85,B 0,C 180,E1 -9984.314,E2 -9984.314} C_VEL
LIN {X 0,Y 425.567,Z 362.097,A -85,B 0,C 180,E1 -9988.109,E2 -9988.109} C_VEL
LIN {X 0,Y 425.594,Z 362.095,A -85,B 0,C 180,E1 -9990.001,E2 -9990.001} C_VEL
LIN {X 0,Y 425.519,Z 362.101,A -85,B 0,C 180,E1 -9992.841,E2 -9992.841} C_VEL
LIN {X 0,Y 425.531,Z 362.107,A -85,B 0,C 180,E1 -9995.688,E2 -9995.688} C_VEL
LIN {X 0,Y 425.412,Z 362.114,A -85,B 0,C 180,E1 -9998.552,E2 -9998.552} C_VEL
LIN {X 0,Y 425.392,Z 362.119,A -85,B 0,C 180,E1 -9999.122,E2 -9999.122} C_VEL
LIN {X 0,Y 424.737,Z 362.205,A -85,B 0,C 180,E1 -9999.912,E2 -9999.912} C_VEL
LIN {X 0,Y 421.901,Z 362.554,A -85,B 0,C 180,E1 -10001.196,E2 -10001.196} C_VEL
LIN {X 0,Y 419.482,Z 362.854,A -85,B 0,C 180,E1 -10002.232,E2 -10002.232} C_VEL
LIN {X 0,Y 418.423,Z 362.987,A -85,B 0,C 180,E1 -10003.033,E2 -10003.033} C_VEL
LIN {X 0,Y 418.327,Z 363.001,A -85,B 0,C 180,E1 -10003.305,E2 -10003.305} C_VEL
LIN {X 0,Y 418.269,Z 363.004,A -85,B 0,C 180,E1 -10006.714,E2 -10006.714} C_VEL
LIN {X 0,Y 418.276,Z 363.008,A -85,B 0,C 180,E1 -10009.791,E2 -10009.791} C_VEL
LIN {X 0,Y 418.234,Z 363.009,A -85,B 0,C 180,E1 -10012.738,E2 -10012.738} C_VEL
LIN {X 0,Y 418.225,Z 363.013,A -85,B 0,C 180,E1 -10015.908,E2 -10015.908} C_VEL
LIN {X 0,Y 418.265,Z 363.008,A -85,B 0,C 180,E1 -10019.163,E2 -10019.163} C_VEL
LIN {X 0,Y 418.264,Z 363.006,A -85,B 0,C 180,E1 -10022.845,E2 -10022.845} C_VEL
LIN {X 0,Y 418.25,Z 363.012,A -85,B 0,C 180,E1 -10026.238,E2 -10026.238} C_VEL
LIN {X 0,Y 418.235,Z 363.016,A -85,B 0,C 180,E1 -10029.685,E2 -10029.685} C_VEL
LIN {X 0,Y 418.24,Z 363.015,A -85,B 0,C 180,E1 -10031.91,E2 -10031.91} C_VEL
LIN {X 0,Y 420.732,Z 373.593,A -85,B 0,C 180,E1 -10034.106,E2 -10034.106} C_VEL
LIN {X 0,Y 428.327,Z 392.654,A -85,B 0,C 180,E1 -10034.973,E2 -10034.973} C_VEL
LIN {X 0,Y 430.088,Z 400.624,A -85,B 0,C 180,E1 -10035.241,E2 -10035.241} C_VEL
LIN {X 0,Y 426.935,Z 539.492,A -85,B 0,C 180,E1 -10037.894,E2 -10037.894} C_VEL
LIN {X 0,Y 426.293,Z 555.188,A -85,B 0,C 180,E1 -10038.387,E2 -10038.387} C_VEL
LIN {X 0,Y 425.509,Z 570,A -85,B 0,C 180,E1 -10039.044,E2 -10039.044} C_VEL
LIN {X 0,Y 424.566,Z 584.254,A -85,B 0,C 180,E1 -10039.868,E2 -10039.868} C_VEL
LIN {X 0,Y 423.54,Z 598.494,A -85,B 0,C 180,E1 -10040.909,E2 -10040.909} C_VEL
LIN {X 0,Y 422.541,Z 610.942,A -85,B 0,C 180,E1 -10042.018,E2 -10042.018} C_VEL
LIN {X 0,Y 421.437,Z 623.82,A -85,B 0,C 180,E1 -10043.41,E2 -10043.41} C_VEL
LIN {X 0,Y 420.356,Z 635.368,A -85,B 0,C 180,E1 -10044.914,E2 -10044.914} C_VEL
LIN {X 0,Y 419.505,Z 645.162,A -85,B 0,C 180,E1 -10046.437,E2 -10046.437} C_VEL
LIN {X 0,Y 418.752,Z 654.039,A -85,B 0,C 180,E1 -10048.084,E2 -10048.084} C_VEL
LIN {X 0,Y 418.087,Z 662.491,A -85,B 0,C 180,E1 -10049.993,E2 -10049.993} C_VEL
LIN {X 0,Y 417.623,Z 669.255,A -85,B 0,C 180,E1 -10051.887,E2 -10051.887} C_VEL
LIN {X 0,Y 417.373,Z 674.105,A -85,B 0,C 180,E1 -10053.602,E2 -10053.602} C_VEL
LIN {X 0,Y 417.092,Z 678.225,A -85,B 0,C 180,E1 -10055.493,E2 -10055.493} C_VEL
LIN {X 0,Y 416.95,Z 680.895,A -85,B 0,C 180,E1 -10057.189,E2 -10057.189} C_VEL
LIN {X 0,Y 416.94,Z 682.064,A -85,B 0,C 180,E1 -10058.233,E2 -10058.233} C_VEL
LIN {X 0,Y 416.872,Z 683.356,A -85,B 0,C 180,E1 -10060.295,E2 -10060.295} C_VEL
LIN {X 0,Y 416.867,Z 683.307,A -85,B 0,C 180,E1 -10062.334,E2 -10062.334} C_VEL
LIN {X 0,Y 416.942,Z 681.959,A -85,B 0,C 180,E1 -10064.353,E2 -10064.353} C_VEL
LIN {X 0,Y 417.063,Z 679.312,A -85,B 0,C 180,E1 -10066.354,E2 -10066.354} C_VEL
LIN {X 0,Y 417.338,Z 675.341,A -85,B 0,C 180,E1 -10068.341,E2 -10068.341} C_VEL
LIN {X 0,Y 417.657,Z 670.021,A -85,B 0,C 180,E1 -10070.312,E2 -10070.312} C_VEL
LIN {X 0,Y 418.329,Z 662.728,A -85,B 0,C 180,E1 -10072.404,E2 -10072.404} C_VEL
LIN {X 0,Y 418.982,Z 654.776,A -85,B 0,C 180,E1 -10074.223,E2 -10074.223} C_VEL
LIN {X 0,Y 419.797,Z 645.774,A -85,B 0,C 180,E1 -10075.92,E2 -10075.92} C_VEL
LIN {X 0,Y 420.959,Z 634.926,A -85,B 0,C 180,E1 -10077.608,E2 -10077.608} C_VEL
LIN {X 0,Y 421.95,Z 623.858,A -85,B 0,C 180,E1 -10079.045,E2 -10079.045} C_VEL
LIN {X 0,Y 423.15,Z 611.756,A -85,B 0,C 180,E1 -10080.357,E2 -10080.357} C_VEL
LIN {X 0,Y 424.381,Z 598.537,A -85,B 0,C 180,E1 -10081.542,E2 -10081.542} C_VEL
LIN {X 0,Y 425.553,Z 583.911,A -85,B 0,C 180,E1 -10082.603,E2 -10082.603} C_VEL
LIN {X 0,Y 426.565,Z 569.548,A -85,B 0,C 180,E1 -10083.424,E2 -10083.424} C_VEL
LIN {X 0,Y 427.399,Z 554.073,A -85,B 0,C 180,E1 -10084.096,E2 -10084.096} C_VEL
LIN {X 0,Y 428.069,Z 538.695,A -85,B 0,C 180,E1 -10084.561,E2 -10084.561} C_VEL
LIN {X 0,Y 431.591,Z 416.957,A -85,B 0,C 180,E1 -10087.062,E2 -10087.062} C_VEL
LIN {X 0,Y 432.068,Z 400.952,A -85,B 0,C 180,E1 -10087.402,E2 -10087.402} C_VEL
LIN {X 0,Y 430.486,Z 394.231,A -85,B 0,C 180,E1 -10087.696,E2 -10087.696} C_VEL
LIN {X 0,Y 423.524,Z 379.352,A -85,B 0,C 180,E1 -10088.666,E2 -10088.666} C_VEL
LIN {X 0,Y 421.809,Z 375.834,A -85,B 0,C 180,E1 -10088.937,E2 -10088.937} C_VEL
LIN {X 0,Y 418.967,Z 365.331,A -85,B 0,C 180,E1 -10091.612,E2 -10091.612} C_VEL
LIN {X 0,Y 418.375,Z 362.998,A -85,B 0,C 180,E1 -10092.244,E2 -10092.244} C_VEL
LIN {X 0,Y 418.306,Z 363.007,A -85,B 0,C 180,E1 -10095.594,E2 -10095.594} C_VEL
LIN {X 0,Y 418.28,Z 363.01,A -85,B 0,C 180,E1 -10098.617,E2 -10098.617} C_VEL
LIN {X 0,Y 418.239,Z 363.012,A -85,B 0,C 180,E1 -10101.696,E2 -10101.696} C_VEL
LIN {X 0,Y 418.248,Z 363.011,A -85,B 0,C 180,E1 -10104.852,E2 -10104.852} C_VEL
LIN {X 0,Y 418.211,Z 363.017,A -85,B 0,C 180,E1 -10108.069,E2 -10108.069} C_VEL
LIN {X 0,Y 418.241,Z 363.01,A -85,B 0,C 180,E1 -10111.018,E2 -10111.018} C_VEL
LIN {X 0,Y 418.235,Z 363.013,A -85,B 0,C 180,E1 -10113.678,E2 -10113.678} C_VEL
LIN {X 0,Y 418.235,Z 363.012,A -85,B 0,C 180,E1 -10117.224,E2 -10117.224} C_VEL
LIN {X 0,Y 418.209,Z 363.015,A -85,B 0,C 180,E1 -10120.866,E2 -10120.866} C_VEL
LIN {X 0,Y 418.203,Z 363.015,A -85,B 0,C 180,E1 -10123.727,E2 -10123.727} C_VEL
LIN {X 0,Y 418.201,Z 363.016,A -85,B 0,C 180,E1 -10126.446,E2 -10126.446} C_VEL
LIN {X 0,Y 418.208,Z 363.014,A -85,B 0,C 180,E1 -10129.132,E2 -10129.132} C_VEL
LIN {X 0,Y 418.234,Z 363.014,A -85,B 0,C 180,E1 -10132.774,E2 -10132.774} C_VEL
LIN {X 0,Y 418.258,Z 363.121,A -85,B 0,C 180,E1 -10135.713,E2 -10135.713} C_VEL
LIN {X 0,Y 421.382,Z 373.864,A -85,B 0,C 180,E1 -10138.277,E2 -10138.277} C_VEL
LIN {X 0,Y 424.108,Z 385.249,A -85,B 0,C 180,E1 -10140.734,E2 -10140.734} C_VEL
LIN {X 0,Y 425.238,Z 391.034,A -85,B 0,C 180,E1 -10141.898,E2 -10141.898} C_VEL
LIN {X 0,Y 425.002,Z 394.097,A -85,B 0,C 180,E1 -10142.4,E2 -10142.4} C_VEL
LIN {X 0,Y 429.091,Z 413.238,A -85,B 0,C 180,E1 -10143.221,E2 -10143.221} C_VEL
LIN {X 0,Y 431.582,Z 428.413,A -85,B 0,C 180,E1 -10143.776,E2 -10143.776} C_VEL
LIN {X 0,Y 428.293,Z 540.676,A -85,B 0,C 180,E1 -10146.069,E2 -10146.069} C_VEL
LIN {X 0,Y 427.636,Z 564.131,A -85,B 0,C 180,E1 -10146.576,E2 -10146.576} C_VEL
LIN {X 0,Y 426.671,Z 579.781,A -85,B 0,C 180,E1 -10147.091,E2 -10147.091} C_VEL
LIN {X 0,Y 425.691,Z 595.174,A -85,B 0,C 180,E1 -10147.81,E2 -10147.81} C_VEL
LIN {X 0,Y 424.622,Z 609.058,A -85,B 0,C 180,E1 -10148.645,E2 -10148.645} C_VEL
LIN {X 0,Y 423.402,Z 623.407,A -85,B 0,C 180,E1 -10149.725,E2 -10149.725} C_VEL
LIN {X 0,Y 422.162,Z 636.478,A -85,B 0,C 180,E1 -10150.93,E2 -10150.93} C_VEL
